(* CODESYS project tc2_bacnetrev12.library
   Company: Beckhoff Automation GmbH
   DefaultNamespace: Tc2_BACnetRev12
   Title: Tc2_BACnetRev12
   Description: The PLC library is a collection of function blocks for programming a BACnet controller. For each BACnet object function blocks are available that are read and written via the selected properties. In general a distinction is made between function blocks for server and client objects. Function blocks for client objects have the prefix "Remote", since they enable access to remote BACnet objects on other devices. The BACnet object function blocks ascertain whether process data are valid and the BACnet controller is ready for operation (bReady).
   Placeholder: Tc2_BACnetRev12
   Author: Beckhoff Automation
   Version: 2.4.3.0

Project tree, tasks and I/O mapping:
  libraries: Tc2_Standard, * (Beckhoff Automation GmbH); Tc2_System, * (Beckhoff Automation GmbH); Tc2_Utilities, * (Beckhoff Automation GmbH)
  Data types/
    BACnet Datatypes/
      [internal]/
        ADS/
          data type ST_BACnet_GlobalAdsBuffer
        CalendarEntry/
          data type E_BACnetCalendarEntryChoice
          data type E_BACnetCalendarEntryType
          data type ST_BACnet_CalendarEntryDate
          data type ST_BACnet_CalendarEntryDateRange
          data type ST_BACnet_CalendarEntryWeekNDay
        ExceptionSchedule/
          data type ST_BACnet_ExceptionScheduleCalDate
          data type ST_BACnet_ExceptionScheduleCalRef
          data type ST_BACnet_ExceptionScheduleCalWnD
        LogRecord/
          data type E_BACnetLogRecordChoice
          data type ST_BACnet_LogDatum
          data type ST_BACnet_LogDatumList
          data type ST_BACnet_LogRecord
          data type ST_BACnet_LogRecordList
        NotificationSink/
          data type ST_BACnet_NotificationSinkEventEntry
          data type ST_BACnet_NSinkEventValidFields
        Recipient/
          data type E_BACnetRecipientChoice
          data type ST_BACnet_DestinationDevice
          data type ST_BACnet_RecipientDevice
          data type T_BACnet_DestinationDeviceArray
        SpecialEvent/
          data type E_BACnetSpecialEventChoice
          data type ST_BACnet_SpecialEventCalendarEntryDate
          data type ST_BACnet_SpecialEventCalendarEntryRange
          data type ST_BACnet_SpecialEventCalendarEntryWnD
          data type ST_BACnet_SpecialEventCalendarReference
          data type ST_BACnet_SpecialEventListCalEntryDate
          data type ST_BACnet_SpecialEventListCalEntryRange
          data type ST_BACnet_SpecialEventListCalEntryWnD
          data type ST_BACnet_SpecialEventListCalReference
        WeeklySchedule/
          data type ST_BACnet_DailySchedule
        data type E_BACnetTimeStampChoice
        data type ST_BACnet_TimeStampDateTime
      [obsolete]/
        data type FB_BACnet_Accumulator_R9
        data type FB_BACnet_AnalogInput_R9
        data type FB_BACnet_AnalogOutput_R9
        data type FB_BACnet_AnalogValue_R9
        data type FB_BACnet_Averaging_R9
        data type FB_BACnet_BinaryInput_R9
        data type FB_BACnet_BinaryOutput_R9
        data type FB_BACnet_BinaryValue_R9
        data type FB_BACnet_Calendar_R9
        data type FB_BACnet_Command_R9
        data type FB_BACnet_Device_R9
        data type FB_BACnet_EventEnrollment_R9
        data type FB_BACnet_File_R9
        data type FB_BACnet_Group_R9
        data type FB_BACnet_Loop_R9
        data type FB_BACnet_MultiStateInput_R9
        data type FB_BACnet_MultiStateOutput_R9
        data type FB_BACnet_MultiStateValue_R9
        data type FB_BACnet_NotificationClass_R9
        data type FB_BACnet_Program_R9
        data type FB_BACnet_PulseConverter_R9
        data type FB_BACnet_Schedule_R9
        data type FB_BACnet_TrendLog_R9
      Diagnose/
        data type ST_BACnet_ConfirmedServiceDiag
        data type ST_BACnet_DiagEthStatistics
        data type ST_BACnet_DiagnosisTiming
        data type ST_BACnet_FrameStatistics
        data type ST_BACnet_Info
        data type ST_BACnet_ServerStatistics
        data type ST_BACnet_TcIoEthStatistic
        data type ST_BACnet_TcIoEthTxRxErrorCount
        data type ST_BACnet_UnConfirmedServiceDiag
      data type ST_BACnet_AdsConnection
      data type ST_BACnet_CharacterStringExt
      data type ST_BACnet_CharacterStringExtListEntry
      data type ST_BACnet_Date
      data type ST_BACnet_DateTime
      data type ST_BACnet_Diagnosis
      data type ST_BACnet_EventTransitionBits
      data type ST_BACnet_ExceptionScheduleBool
      data type ST_BACnet_ExceptionScheduleEntryBool
      data type ST_BACnet_ExceptionScheduleEntryReal
      data type ST_BACnet_ExceptionScheduleReal
      data type ST_BACnet_LimitEnable
      data type ST_BACnet_LogBufferEntryReal
      data type ST_BACnet_LogBufferReal
      data type ST_BACnet_NSinkEvent
      data type ST_BACnet_ObjectIdentifierList
      data type ST_BACnet_ObjectTypesSupported
      data type ST_BACnet_ProgramHandshakeRequests
      data type ST_BACnet_ProgramHandshakeStates
      data type ST_BACnet_RecipientListDevice
      data type ST_BACnet_RecipientListDeviceEntry
      data type ST_BACnet_ServicesSupported
      data type ST_BACnet_StatusFlags
      data type ST_BACnet_Time
      data type ST_BACnet_TimeValue
      data type ST_BACnet_TimeValueBool
      data type ST_BACnet_TimeValueList
      data type ST_BACnet_TimeValueReal
      data type ST_BACnet_Value
      data type ST_BACnet_WeeklyScheduleBool
      data type ST_BACnet_WeeklyScheduleReal
      data type T_BACnet_CalendarEntryTypeFilter
      data type T_BACnet_ObjectIdentifier
    BACnet Enumerations/
      data type E_BACNETACTION
      data type E_BACNETADAPTERSTATUS
      data type E_BACNETBINARYPV
      data type E_BACNETDATATYPES
      data type E_BACNETDAYSOFWEEKBITS
      data type E_BACNETDEVICESTATUS
      data type E_BACNETEVENTSTATE
      data type E_BACNETEVENTTRANSITIONBIT
      data type E_BACNETEVENTTYPE
      data type E_BACNETFILEACCESSMETHOD
      data type E_BACNETLIFESAFETYMODE
      data type E_BACNETLIFESAFETYOPERATION
      data type E_BACNETLIMITENABLEBITS
      data type E_BACNETLOGGINGTYPE
      data type E_BACNETLOOPMODE
      data type E_BACNETNOTIFYTYPE
      data type E_BACNETOBJECTSUPPORTEDBITS
      data type E_BACNETOBJECTTYPE
      data type E_BACNETPERSISTENTDATASTATE
      data type E_BACNETPIDTUNINGMODE
      data type E_BACNETPOLARITY
      data type E_BACNETPRIORITY
      data type E_BACNETPROGRAMERROR
      data type E_BACNETPROGRAMREQUEST
      data type E_BACNETPROGRAMSTATE
      data type E_BACNETPROPERTYIDENTIFIER
      data type E_BACNETRELIABILITY
      data type E_BACNETSEGMENTATION
      data type E_BACNETSERVICESSUPPORTEDBITS
      data type E_BACNETSILENCEDSTATE
      data type E_BACNETSTATUSFLAGS
      data type E_BACNETSTRINGENCODINGTYPES
      data type E_BACNETUNIT
  Global Variables/
    global variables BACnet_Globals
  POUs/
    [obsolete]/
      function F_GetVersionTcBACnet [ST]
    BACnet ADS/
      [obsolete]/
        function block FB_BACnet_NotificationSinkDelEntry [ST]
      Connection/
        function block _FB_BACnet_AdsConn [ST]
      Properties/
        Common/
          function block FB_BACnet_ReadProp [ST]
          function block FB_BACnet_WriteProp [ST]
        function block FB_BACnet_DescriptionProperty [ST]
        function block FB_BACnet_EventMessageTextsProperty [ST]: _NextEntry
        function block FB_BACnet_ExceptionScheduleProperty [ST]: _NextEvent, _NextTimeValue
        function block FB_BACnet_ExceptionSchedulePropertyReal [ST]: _NextEvent, _NextTimeValue
        function block FB_BACnet_LogBufferProperty [ST]: _NextLogDatum, _NextLogRecord
        function block FB_BACnet_ObjectListProperty [ST]
        function block FB_BACnet_ObjectNameProperty [ST]
        function block FB_BACnet_RecipientListProperty [ST]
        function block FB_BACnet_WeeklyScheduleProperty [ST]: _NextDay, _NextTimeValue
        function block FB_BACnet_WeeklySchedulePropertyReal [ST]: _NextDay, _NextTimeValue
      function block FB_BACnet_GetDiagInfo [ST]
      function block FB_BACnet_NSinkAcknEvent [ST]
      function block FB_BACnet_NSinkReadEvent [ST]
      function block FB_BACnet_NSinkRemoveEvent [ST]
      function block FB_BACnet_TimeSync [ST]
    BACnet Helper/
      [internal]/
        function _F_BACnet_AlignedSize [ST]
        function _F_BACnet_BitFieldBit [ST]
        function _F_BACnet_ChangeBitFieldBit [ST]
        function _F_BACnet_ChrStrExtLen [ST]
        function _F_BACnet_DecodeUCS2 [ST]
        function _F_BACnet_DecodeUCS4 [ST]
        function _F_BACnet_DecodeUTF8 [ST]
        function _F_BACnet_EncodeUTF8 [ST]
        function _F_BACnet_IsBitFieldBitSet [ST]
        function _F_BACnet_SetBitFieldBit [ST]
        function _F_BACnet_SysTimeDiff [ST]
        function _F_BACnet_UCS2ToWin1252 [ST]
        function _F_BACnet_UnSetBitFieldBit [ST]
        function _F_BACnet_Utf8ToWin1252 [ST]
        function _F_BACnet_Win1252ToUCS2 [ST]
        function _F_BACnet_Win1252ToUtf8 [ST]
        function block _FB_BACnet_PidTune [ST]
        function F_BACnet_AnalogPV [ST]
      DateTime/
        function F_BACnet_CheckDay [ST]
        function F_BACnet_CheckDayOfWeek [ST]
        function F_BACnet_CheckHour [ST]
        function F_BACnet_CheckHundredths [ST]
        function F_BACnet_CheckMinute [ST]
        function F_BACnet_CheckMonth [ST]
        function F_BACnet_CheckSecond [ST]
        function F_BACnet_CheckWeekOfMonth [ST]
        function F_BACnet_CheckYear [ST]
        function F_BACnet_DateHasPlaceholder [ST]
        function F_BACnet_DateMerge [ST]
        function F_BACnet_DateTime_TO_TimeStruct [ST]
        function F_BACnet_DateTimeString [ST]
        function F_BACnet_DateUnspecified [ST]
        function F_BACnet_DaysInMonth [ST]
        function F_BACnet_Get100msDate [ST]
        function F_BACnet_Get100msTime [ST]
        function F_BACnet_TimeHasPlaceholder [ST]
        function F_BACnet_TimeMerge [ST]
        function F_BACnet_TimeString [ST]
        function F_BACnet_TimeStruct_TO_DateTime [ST]
        function F_BACnet_TimeUnspecified [ST]
      Flags/
        function F_BACnet_EventTransitionFlags [ST]
        function F_BACnet_GetEventTransFlagsData [ST]
        function F_BACnet_GetLimitEnFlagsData [ST]
        function F_BACnet_GetStatusFlagsData [ST]
        function F_BACnet_LimitEnableFlags [ST]
        function F_BACnet_StatusFlags [ST]
      MultiState/
        function F_BACnet_MultiStatePV [ST]
      Real/
        function F_BACnet_IsFinite [ST]
        function F_BACnet_NAN [ST]
        function F_BACnet_RealEQ [ST]
        function F_BACnet_RealGE [ST]
        function F_BACnet_RealGT [ST]
        function F_BACnet_RealLE [ST]
        function F_BACnet_RealLT [ST]
        function F_BACnet_RealNothing [ST]
        function F_BACnet_RealNull [ST]
        function F_BACnet_RealPV [ST]
        function F_BACnet_RealToStr [ST]
      String/
        function F_BACnet_GetObjectIdString [ST]
        function block FB_BACnet_StringExtDecode [ST]
        function block FB_BACnet_StringExtEncode [ST]
      function F_BACnet_GetObjectListIndex [ST]
      function F_BACnet_GetObjId [ST]
      function F_BACnet_GetObjInstance [ST]
      function F_BACnet_GetObjType [ST]
      function block FB_BACnet_AccLimit [ST]
      function block FB_BACnet_AvgValue [ST]
      function block FB_BACnet_PidControl [ST]
      function block FB_BACnet_PT1 [ST]
    BACnet Logic/
      function F_BinPV_AND [ST]
      function F_BinPV_NOT [ST]
      function F_BinPV_OR [ST]
      function F_BinPV_To_Bool [ST]
      function F_BinPV_XOR [ST]
      function F_Bool_To_BinPV [ST]
    BACnet Objects/
      Local (Server)/
        [Internal]/
          function block _FB_BACnet_AnalogObject [ST]
          function block _FB_BACnet_BinaryObject [ST]
          function block _FB_BACnet_Object [ST]
        ADS/
          function block FB_BACnet_AnalogOutput_ADS [ST]
          function block FB_BACnet_AnalogValue_ADS [ST]
          function block FB_BACnet_BinaryOutput_ADS [ST]
          function block FB_BACnet_BinaryValue_ADS [ST]
          function block FB_BACnet_MultiStateOutput_ADS [ST]
          function block FB_BACnet_MultiStateValue_ADS [ST]
        DRV/
          function block FB_BACnet_Loop_DRV [ST]
          function block FB_BACnet_Loop_DRV_EX [ST]
        Extended Process Data/
          function block FB_BACnet_Accumulator_EX [ST]
          function block FB_BACnet_AnalogInput_EX [ST]
          function block FB_BACnet_AnalogOutput_EX [ST]
          function block FB_BACnet_AnalogValue_EX [ST]
          function block FB_BACnet_Averaging_EX [ST]
          function block FB_BACnet_BinaryInput_EX [ST]
          function block FB_BACnet_BinaryOutput_EX [ST]
          function block FB_BACnet_BinaryValue_EX [ST]
          function block FB_BACnet_Calendar_EX [ST]
          function block FB_BACnet_Command_EX [ST]
          function block FB_BACnet_EventEnrollment_EX [ST]
          function block FB_BACnet_File_EX [ST]
          function block FB_BACnet_Group_EX [ST]
          function block FB_BACnet_Loop_EX [ST]
          function block FB_BACnet_MultiStateInput_EX [ST]
          function block FB_BACnet_MultiStateOutput_EX [ST]
          function block FB_BACnet_MultiStateValue_EX [ST]
          function block FB_BACnet_NotificationClass_EX [ST]
          function block FB_BACnet_Program_EX [ST]
          function block FB_BACnet_PulseConverter_EX [ST]
          function block FB_BACnet_Schedule_EX [ST]
          function block FB_BACnet_TrendLog_EX [ST]
        R6/
          function block FB_BACnet_Accumulator_R6 [ST]
          function block FB_BACnet_Accumulator_RAW_R6 [ST]
        RAW/
          function block FB_BACnet_Accumulator_RAW [ST]
          function block FB_BACnet_AnalogInput_RAW [ST]
          function block FB_BACnet_AnalogOutput_RAW [ST]
          function block FB_BACnet_BinaryInput_RAW [ST]
          function block FB_BACnet_BinaryOutput_RAW [ST]
          function block FB_BACnet_MultiStateInput_RAW [ST]
          function block FB_BACnet_MultiStateOutput_RAW [ST]
          function block FB_BACnet_PulseConverter_RAW [ST]
        function block FB_BACnet_Accumulator [ST]
        function block FB_BACnet_AnalogInput [ST]
        function block FB_BACnet_AnalogOutput [ST]
        function block FB_BACnet_AnalogValue [ST]
        function block FB_BACnet_Averaging [ST]
        function block FB_BACnet_BinaryInput [ST]
        function block FB_BACnet_BinaryOutput [ST]
        function block FB_BACnet_BinaryValue [ST]
        function block FB_BACnet_Calendar [ST]
        function block FB_BACnet_Command [ST]
        function block FB_BACnet_Device [ST]
        function block FB_BACnet_EventEnrollment [ST]
        function block FB_BACnet_File [ST]
        function block FB_BACnet_Group [ST]
        function block FB_BACnet_Loop [ST]
        function block FB_BACnet_MultiStateInput [ST]
        function block FB_BACnet_MultiStateOutput [ST]
        function block FB_BACnet_MultiStateValue [ST]
        function block FB_BACnet_NotificationClass [ST]
        function block FB_BACnet_Program [ST]
        function block FB_BACnet_PulseConverter [ST]
        function block FB_BACnet_Schedule [ST]
        function block FB_BACnet_TrendLog [ST]
      Remote (Client)/
        Extended Process Data/
          function block FB_BACnet_RemoteAccumulator_EX [ST]
          function block FB_BACnet_RemoteAnalogInput_EX [ST]
          function block FB_BACnet_RemoteAnalogOutput_EX [ST]
          function block FB_BACnet_RemoteAnalogValue_EX [ST]
          function block FB_BACnet_RemoteAveraging_EX [ST]
          function block FB_BACnet_RemoteBinaryInput_EX [ST]
          function block FB_BACnet_RemoteBinaryOutput_EX [ST]
          function block FB_BACnet_RemoteBinaryValue_EX [ST]
          function block FB_BACnet_RemoteCalendar_EX [ST]
          function block FB_BACnet_RemoteCommand_EX [ST]
          function block FB_BACnet_RemoteEventEnrollment_EX [ST]
          function block FB_BACnet_RemoteFile_EX [ST]
          function block FB_BACnet_RemoteGroup_EX [ST]
          function block FB_BACnet_RemoteLoop_EX [ST]
          function block FB_BACnet_RemoteMultiStateInput_EX [ST]
          function block FB_BACnet_RemoteMultiStateOutput_EX [ST]
          function block FB_BACnet_RemoteMultiStateValue_EX [ST]
          function block FB_BACnet_RemoteNotificationClass_EX [ST]
          function block FB_BACnet_RemoteProgram_EX [ST]
          function block FB_BACnet_RemotePulseConverter_EX [ST]
          function block FB_BACnet_RemoteSchedule_EX [ST]
          function block FB_BACnet_RemoteTrendLog_EX [ST]
        WRITE/
          function block FB_BACnet_RemoteAnalogOutput_WR [ST]
          function block FB_BACnet_RemoteAnalogValue_WR [ST]
          function block FB_BACnet_RemoteBinaryOutput_WR [ST]
          function block FB_BACnet_RemoteBinaryValue_WR [ST]
          function block FB_BACnet_RemoteCommand_WR [ST]
          function block FB_BACnet_RemoteMultiStateOutput_WR [ST]
          function block FB_BACnet_RemoteMultiStateValue_WR [ST]
          function block FB_BACnet_RemoteProgram_WR [ST]
        function block FB_BACnet_RemoteAccumulator [ST]
        function block FB_BACnet_RemoteAnalogInput [ST]
        function block FB_BACnet_RemoteAnalogOutput [ST]
        function block FB_BACnet_RemoteAnalogValue [ST]
        function block FB_BACnet_RemoteAveraging [ST]
        function block FB_BACnet_RemoteBinaryInput [ST]
        function block FB_BACnet_RemoteBinaryOutput [ST]
        function block FB_BACnet_RemoteBinaryValue [ST]
        function block FB_BACnet_RemoteCalendar [ST]
        function block FB_BACnet_RemoteCommand [ST]
        function block FB_BACnet_RemoteDevice [ST]
        function block FB_BACnet_RemoteEventEnrollment [ST]
        function block FB_BACnet_RemoteFile [ST]
        function block FB_BACnet_RemoteGroup [ST]
        function block FB_BACnet_RemoteLoop [ST]
        function block FB_BACnet_RemoteMultiStateInput [ST]
        function block FB_BACnet_RemoteMultiStateOutput [ST]
        function block FB_BACnet_RemoteMultiStateValue [ST]
        function block FB_BACnet_RemoteNotificationClass [ST]
        function block FB_BACnet_RemoteProgram [ST]
        function block FB_BACnet_RemotePulseConverter [ST]
        function block FB_BACnet_RemoteSchedule [ST]
        function block FB_BACnet_RemoteTrendLog [ST]
    BACnet Signals/
      function block FB_BACnet_PWM [ST]
    function block FB_BACnet_Adapter [ST]: UpdateNetID
    function block FB_BACnet_NotificationSink [ST]
  Version/
    global variables Global_Version
*)

// Data types/BACnet Datatypes/[internal]/ADS/ST_BACnet_GlobalAdsBuffer
TYPE ST_BACnet_GlobalAdsBuffer :
STRUCT
	bTestSet	: BOOL;
	iLocked		: DINT; (* -1 Buffer not ready, 0 Buffer ready, 1..n Buffer used (locked) *)
	arrData		: ARRAY[0..BACnet_ADSBufferSize] OF BYTE;
END_STRUCT
END_TYPE

// Data types/BACnet Datatypes/[internal]/CalendarEntry/E_BACnetCalendarEntryChoice
TYPE E_BACnetCalendarEntryChoice :
(
(*
	BACnetDate              DATE;
	BACnetDateRange   		dateRange;
	BACnetWeekNDay          weekNDay;
*)
	BACnetCalendarEntryChoice_date,
	BACnetCalendarEntryChoice_dateRange,
	BACnetCalendarEntryChoice_weekNDay
);
END_TYPE

// Data types/BACnet Datatypes/[internal]/CalendarEntry/E_BACnetCalendarEntryType
TYPE E_BACnetCalendarEntryType : (* Not a BACnet-Stack type! *)
(
	BACnetCalendarEntryType_None,
	BACnetCalendarEntryType_Ref,
	BACnetCalendarEntryType_Date,
	BACnetCalendarEntryType_DateRange,
	BACnetCalendarEntryType_WeekNDay
);
END_TYPE

// Data types/BACnet Datatypes/[internal]/CalendarEntry/ST_BACnet_CalendarEntryDate
TYPE ST_BACnet_CalendarEntryDate :
STRUCT
(*
	typedef struct _BACnetCalendarEntry
	{
	      BACnetCalendarEntryChoice choice;
	      union
	      {
	            BACnetDate              date;
	            BACnetDateRange   dateRange;
	            BACnetWeekNDay          weekNDay;
	      };
	}BACnetCalendarEntry, *PBACnetCalendarEntry;
*)
	eEntryChoice		: E_BACnetCalendarEntryChoice;
	nRes				: WORD; (* ENUM alignment *)
	stDate				: ST_BACnet_Date;
END_STRUCT
END_TYPE

// Data types/BACnet Datatypes/[internal]/CalendarEntry/ST_BACnet_CalendarEntryDateRange
TYPE ST_BACnet_CalendarEntryDateRange :
STRUCT
(*
	typedef struct _BACnetCalendarEntry
	{
	      BACnetCalendarEntryChoice choice;
	      union
	      {
	            BACnetDate              date;
	            BACnetDateRange   dateRange;
	            BACnetWeekNDay          weekNDay;
	      };
	}BACnetCalendarEntry, *PBACnetCalendarEntry;
*)
	eEntryChoice		: E_BACnetCalendarEntryChoice;
	nRes				: WORD; (* ENUM alignment *)
	stStartDate			: ST_BACnet_Date;
	stEndDate			: ST_BACnet_Date;
END_STRUCT
END_TYPE

// Data types/BACnet Datatypes/[internal]/CalendarEntry/ST_BACnet_CalendarEntryWeekNDay
TYPE ST_BACnet_CalendarEntryWeekNDay :
STRUCT
(*
	typedef struct _BACnetCalendarEntry
	{
	      BACnetCalendarEntryChoice choice;
	      union
	      {
	            BACnetDate              date;
	            BACnetDateRange   dateRange;
	            BACnetWeekNDay          weekNDay;
	      };
	}BACnetCalendarEntry, *PBACnetCalendarEntry;
*)
	eEntryChoice	: E_BACnetCalendarEntryChoice;
	nRes1			: WORD; (* ENUM alignment *)
	iMonth			: USINT;
	iWeekOfMonth	: USINT;
	iDay			: USINT;
	nRes2			: USINT; (* weekNDay alignment *)
END_STRUCT
END_TYPE

// Data types/BACnet Datatypes/[internal]/ExceptionSchedule/ST_BACnet_ExceptionScheduleCalDate
TYPE ST_BACnet_ExceptionScheduleCalDate :
STRUCT
	stStart			: ST_BACnet_Date;
	stEnd			: ST_BACnet_Date;
END_STRUCT
END_TYPE

// Data types/BACnet Datatypes/[internal]/ExceptionSchedule/ST_BACnet_ExceptionScheduleCalRef
TYPE ST_BACnet_ExceptionScheduleCalRef :
STRUCT
	tCalObjectId	: T_BACnet_ObjectIdentifier := 16#FFFFFFFF;
END_STRUCT
END_TYPE

// Data types/BACnet Datatypes/[internal]/ExceptionSchedule/ST_BACnet_ExceptionScheduleCalWnD
TYPE ST_BACnet_ExceptionScheduleCalWnD :
STRUCT
	iMonth			: USINT; (* 255 = all months of year *)
	iWeekOfMonth	: USINT; (* 255 = all weeks of month *)
	iDay			: USINT; (* 255 = all days of month *)
END_STRUCT
END_TYPE

// Data types/BACnet Datatypes/[internal]/LogRecord/E_BACnetLogRecordChoice
TYPE E_BACnetLogRecordChoice :
(
(*
enum BACnetLogRecordChoice
{
      logStatus,              // [0] BACnetLogStatus,
      booleanValue,           // [1] BOOL,
      realValue,              // [2] REAL,
      enumValue,              // [3] ENUMERATED, __ Optionally limited to 32 bits
      unsignedValue,          // [4] Unsigned, __ Optionally limited to 32 bits
      signedValue,            // [5] INTEGER, __ Optionally limited to 32 bits
      bitstringValue,         // [6] BIT STRING, __ Optionally limited to 32 bits
      nullValue,              // [7] NULL,
      failure,                // [8] Error,
      timeChange,             // [9] REAL,
      anyValue,               // [10] ABSTRACT_SYNTAX.&Type __ Optional
};
*)
	BACnetLogRecordChoice_logStatus 	:= 0, (* BACnetLogStatus *)
	BACnetLogRecordChoice_booleanValue := 1, (*  BOOL, *)
	BACnetLogRecordChoice_realValue	:= 2, (*  REAL, *)
	BACnetLogRecordChoice_enumValue	:= 3, (*  ENUMERATED, __ Optionally limited TO 32 bits *)
	BACnetLogRecordChoice_unsignedValue:= 4, (*  Unsigned, __ Optionally limited TO 32 bits *)
	BACnetLogRecordChoice_signedValue	:= 5, (*  INTEGER, __ Optionally limited TO 32 bits *)
	BACnetLogRecordChoice_bitstringValue:= 6, (*  BIT STRING, __ Optionally limited TO 32 bits *)
	BACnetLogRecordChoice_nullValue	:= 7, (*  NULL, *)
	BACnetLogRecordChoice_failure		:= 8, (*  Error, *)
	BACnetLogRecordChoice_timeChange	:= 9, (*  REAL, *)
	BACnetLogRecordChoice_anyValue		:= 10 (*  ABSTRACT_SYNTAX.&TYPE __ Optional *)
);
END_TYPE

// Data types/BACnet Datatypes/[internal]/LogRecord/ST_BACnet_LogDatum
TYPE ST_BACnet_LogDatum :
STRUCT
(*

typedef struct _BACnetLogDatum
{
      BACnetLogRecordChoice choice;
      union
      {
            DWORD logStatus; // BitString ... of type BACnetLogStatus
            BOOL booleanValue;
            FLOAT realValue;
            EnumerationValueType enumerationValue;
            ULONG unsignedValue;
            DWORD signedValue;
            DWORD bitstringValue;
            DWORD nullValue;
            BACnetError failure; 
            FLOAT timeChange;
            AnyType anyValue; // ABSTRACT-SYNTAX.&Type
      };
}BACnetLogDatum, *PBACnetLogDatum;

*)
	choice	: E_BACnetLogRecordChoice;
	nRes	: WORD; (* ENUM alignment to 4 byte *)
	nData	: ARRAY[0..4] OF DWORD; (* 20 byte min. size - data type depending on choice selection *)
END_STRUCT
END_TYPE

// Data types/BACnet Datatypes/[internal]/LogRecord/ST_BACnet_LogDatumList
TYPE ST_BACnet_LogDatumList :
STRUCT
(*

typedef struct _BACnetLogDatumList
{
      DWORD nEntrySize; // 0x80000000 -> next entry
      DWORD reserved;
      BACnetLogDatum listEntry;
}BACnetLogDatumList, *PBACnetLogDatumList;

*)
	nEntrySize	: DWORD; (* 0x80000000 -> next entry *)
	reserved	: DWORD;
	listEntry	: ST_BACnet_LogDatum; (* first entry of log datum list *)
END_STRUCT
END_TYPE

// Data types/BACnet Datatypes/[internal]/LogRecord/ST_BACnet_LogRecord
TYPE ST_BACnet_LogRecord :
STRUCT
(*

typedef STRUCT _BACnetLogRecord
{
      ULONG validFields;
      BACnetDateTime timestamp;          // [0]
      DWORD statusFlags;                       // [2] optional
      BACnetLogDatumList logDatum;  // [1]
}BACnetLogRecord, *PBACnetLogRecord;

*)
	validFields	: UDINT;
	timestamp	: ST_BACnet_DateTime;
	statusFlags	: DWORD;
	logDatum	: ST_BACnet_LogDatumList;
END_STRUCT
END_TYPE

// Data types/BACnet Datatypes/[internal]/LogRecord/ST_BACnet_LogRecordList
TYPE ST_BACnet_LogRecordList :
STRUCT
(*

typedef struct _BACnetLogRecordList
{
      DWORD nEntrySize; // 0x80000000 -> next entry
      DWORD nSequence;  // "reserved"     -> Number of Sequence begins with 1
      BACnetLogRecord listEntry;
}BACnetLogRecordList, *PBACnetLogRecordList;

*)
	nEntrySize	: DWORD; (* 16#80000000 -> next entry *)
	nSequence	: DWORD; (* "reserved"  -> Number OF Sequence begins with 1 *)
	listEntry	: ST_BACnet_LogRecord; (* first entry of record list *)
END_STRUCT
END_TYPE

// Data types/BACnet Datatypes/[internal]/NotificationSink/ST_BACnet_NotificationSinkEventEntry
TYPE ST_BACnet_NotificationSinkEventEntry :
STRUCT
	_fillBytes00				: ARRAY[0..7] OF BYTE; (* list header *)
	validFields					: UDINT;	(*	ULONG validFields; *)
	processIdentifier			: UDINT; (*     ULONG processIdentifier; *)
	initiatingDeviceIdentifier	: T_BACnet_ObjectIdentifier; (*  BACnetObjectIdentifier initiatingDeviceIdentifier; *)
	eventObjectIdentifier		: T_BACnet_ObjectIdentifier; (*  BACnetObjectIdentifier eventObjectIdentifier; *)
	timeStamp					: ST_BACnet_TimeStampDateTime;   (* BACnetTimeStamp timeStamp; *)
	notificationClass			: UDINT;  (* ULONG notificationClass;*)
	priority					: UDINT;  (* ULONG priority; *)
	eventType					: E_BACNETEVENTTYPE; (*  BACnetEventType eventType; *)
	_fillBytes01				: WORD; (* fill bytes *)
	messageText					: ARRAY[1..BACnet_STRING_MAXLENGTH] OF BYTE;
	notifyType					: E_BACNETNOTIFYTYPE;  (* BACnetNotifyType notifyType; *)
	_fillBytes02				: WORD; (* fill bytes *)
	ackRequired					: BOOL; (*  BOOL ackRequired; *)
	_fillBytes03				: ARRAY[0..2] OF BYTE; (* fill bytes *)
	fromState					: E_BACNETEVENTSTATE; (*   BACnetEventState fromState; *)
	_fillBytes04				: WORD; (* fill bytes *)
	toState						: E_BACNETEVENTSTATE; (*  BACnetEventState toState; *)
	_fillBytes05				: WORD; (* fill bytes *)
	eventParameterRaw			: ARRAY[0..127] OF BYTE; (* PBACnetNotificationParameters pEventValues; *)
END_STRUCT
END_TYPE

// Data types/BACnet Datatypes/[internal]/NotificationSink/ST_BACnet_NSinkEventValidFields
TYPE ST_BACnet_NSinkEventValidFields :
STRUCT
      bProcessIdentifier:BOOL; (* Bit0 *)
      bInitiatingDeviceIdentifier:BOOL; (* Bit1 *)
      bEventObjectIdentifier:BOOL; (* Bit2 *)
      bTimeStamp:BOOL; (* Bit3 *)
      bNotificationClass:BOOL; (* Bit4 *)
      bPriority:BOOL; (* Bit5 *)
      bEventType:BOOL; (* Bit6 *)
      bMessageText:BOOL; (* Bit7 *)
      bNotifyType:BOOL; (* Bit8 *)
      bAckRequired:BOOL; (* Bit9 *)
      bFromState:BOOL; (* Bit10 *)
      bToState:BOOL; (* Bit11 *)
      bEventValues:BOOL; (* Bit12 *)
END_STRUCT
END_TYPE

// Data types/BACnet Datatypes/[internal]/Recipient/E_BACnetRecipientChoice
TYPE E_BACnetRecipientChoice :
(
	BACnetRecipientChoice_device,
	BACnetRecipientChoice_address
);
END_TYPE

// Data types/BACnet Datatypes/[internal]/Recipient/ST_BACnet_DestinationDevice
TYPE ST_BACnet_DestinationDevice :
STRUCT
	nValidDaysFlags	: DWORD; (* Bit: 9 = Sunday, 10 = Saturday, 11 = Friday, 12 = Thursday, 13 = Wednesday, 14 = Tuesday, 15 = Monday *)
	stFromTime		: ST_BACnet_Time;
	stToTime		: ST_BACnet_Time;
	stRecipient		: ST_BACnet_RecipientDevice;
	res1			: ARRAY[0..11] OF BYTE; (* allignment *)
	nProcessId		: UDINT;
	nEventTransBits	: DWORD; (* Bit: 12 = to_offnormal, 13 = to_fault, 14 = to_normal *)
	bIssueConfNot	: BOOL;
	res2			: ARRAY[0..2] OF BYTE; (* allignment *)
END_STRUCT
END_TYPE

// Data types/BACnet Datatypes/[internal]/Recipient/ST_BACnet_RecipientDevice
TYPE ST_BACnet_RecipientDevice :
STRUCT
	eRecipientChoice: E_BACnetRecipientChoice;
	res				: WORD; (* allignment *)
	tDeviceId		: T_BACnet_ObjectIdentifier := 16#FFFFFFFF;
END_STRUCT
END_TYPE

// Data types/BACnet Datatypes/[internal]/Recipient/T_BACnet_DestinationDeviceArray
TYPE T_BACnet_DestinationDeviceArray : ARRAY[0..BACnet_MaxDestinationArray] OF ST_BACnet_DestinationDevice; END_TYPE

// Data types/BACnet Datatypes/[internal]/SpecialEvent/E_BACnetSpecialEventChoice
TYPE E_BACnetSpecialEventChoice :
(
(*
	enum BACnetSpecialEventChoice
	{
	      calendarEntry,
	      calendarReference,
	      MaxBACnetSpecialEventChoice
	};
*)
	BACnetSpecialEventChoice_calendarEntry,
	BACnetSpecialEventChoice_calendarReference
);
END_TYPE

// Data types/BACnet Datatypes/[internal]/SpecialEvent/ST_BACnet_SpecialEventCalendarEntryDate
TYPE ST_BACnet_SpecialEventCalendarEntryDate :
STRUCT
(*
	typedef struct _BACnetSpecialEvent
	{
	      BACnetSpecialEventChoice choice;
	      union
	      {
	            BACnetCalendarEntry calendarEntry;
	            BACnetObjectIdentifier calendarReference;
	      };
	      DWORD eventPriority; // DWORD due to alignment
	      DWORD reserved;
	      BACnetTimeValueList listOfTimeValues;
	}BACnetSpecialEvent, *PBACnetSpecialEvent;
*)

	eEventChoice		: E_BACnetSpecialEventChoice;
	nRes1				: WORD; (* ENUM alignment *)
	stCalEntry			: ST_BACnet_CalendarEntryDate;
	nRes2				: DWORD;
	iEventPriority		: DWORD;
	nRes3				: DWORD;
	stListOfTimeValues	: ST_BACnet_TimeValueList;

END_STRUCT
END_TYPE

// Data types/BACnet Datatypes/[internal]/SpecialEvent/ST_BACnet_SpecialEventCalendarEntryRange
TYPE ST_BACnet_SpecialEventCalendarEntryRange :
STRUCT
(*
	typedef struct _BACnetSpecialEvent
	{
	      BACnetSpecialEventChoice choice;
	      union
	      {
	            BACnetCalendarEntry calendarEntry;
	            BACnetObjectIdentifier calendarReference;
	      };
	      DWORD eventPriority; // DWORD due to alignment
	      DWORD reserved;
	      BACnetTimeValueList listOfTimeValues;
	}BACnetSpecialEvent, *PBACnetSpecialEvent;
*)

	eEventChoice		: E_BACnetSpecialEventChoice;
	nRes1				: WORD; (* ENUM alignment *)
	stCalEntry			: ST_BACnet_CalendarEntryDateRange;
	iEventPriority		: DWORD;
	nRes2				: DWORD;
	stListOfTimeValues	: ST_BACnet_TimeValueList;

END_STRUCT
END_TYPE

// Data types/BACnet Datatypes/[internal]/SpecialEvent/ST_BACnet_SpecialEventCalendarEntryWnD
TYPE ST_BACnet_SpecialEventCalendarEntryWnD :
STRUCT
(*
	typedef struct _BACnetSpecialEvent
	{
	      BACnetSpecialEventChoice choice;
	      union
	      {
	            BACnetCalendarEntry calendarEntry;
	            BACnetObjectIdentifier calendarReference;
	      };
	      DWORD eventPriority; // DWORD due to alignment
	      DWORD reserved;
	      BACnetTimeValueList listOfTimeValues;
	}BACnetSpecialEvent, *PBACnetSpecialEvent;
*)

	eEventChoice		: E_BACnetSpecialEventChoice;
	nRes1				: WORD; (* ENUM alignment *)
	stCalEntry			: ST_BACnet_CalendarEntryWeekNDay;
	nRes2				: DWORD;
	iEventPriority		: DWORD;
	nRes3				: DWORD;
	stListOfTimeValues	: ST_BACnet_TimeValueList;

END_STRUCT
END_TYPE

// Data types/BACnet Datatypes/[internal]/SpecialEvent/ST_BACnet_SpecialEventCalendarReference
TYPE ST_BACnet_SpecialEventCalendarReference :
STRUCT
(*
	typedef struct _BACnetSpecialEvent
	{
	      BACnetSpecialEventChoice choice;
	      union
	      {
	            BACnetCalendarEntry calendarEntry;
	            BACnetObjectIdentifier calendarReference;
	      };
	      DWORD eventPriority; // DWORD due to alignment
	      DWORD reserved;
	      BACnetTimeValueList listOfTimeValues;
	}BACnetSpecialEvent, *PBACnetSpecialEvent;
*)

	eEventChoice		: E_BACnetSpecialEventChoice;
	nRes1				: WORD; (* ENUM alignment *)
	tCalRef				: T_BACnet_ObjectIdentifier := 16#FFFFFFFF;
	nRes2				: DWORD;
	nRes3				: DWORD;
	iEventPriority		: DWORD;
	nRes4				: DWORD;
	stListOfTimeValues	: ST_BACnet_TimeValueList;

END_STRUCT
END_TYPE

// Data types/BACnet Datatypes/[internal]/SpecialEvent/ST_BACnet_SpecialEventListCalEntryDate
TYPE ST_BACnet_SpecialEventListCalEntryDate :
STRUCT
(*
	typedef struct _BACnetSpecialEventList
	{
	      DWORD nEntrySize; // 0x80000000 -> next entry
	      DWORD reserved;
	      BACnetSpecialEvent listEntry;
	}BACnetSpecialEventList, *PBACnetSpecialEventList;
*)
	nEntrySize		: DWORD;
	nRes			: DWORD;
	stListEntry		: ST_BACnet_SpecialEventCalendarEntryDate;
END_STRUCT
END_TYPE

// Data types/BACnet Datatypes/[internal]/SpecialEvent/ST_BACnet_SpecialEventListCalEntryRange
TYPE ST_BACnet_SpecialEventListCalEntryRange :
STRUCT
(*
	typedef struct _BACnetSpecialEventList
	{
	      DWORD nEntrySize; // 0x80000000 -> next entry
	      DWORD reserved;
	      BACnetSpecialEvent listEntry;
	}BACnetSpecialEventList, *PBACnetSpecialEventList;
*)
	nEntrySize		: DWORD;
	nRes			: DWORD;
	stListEntry		: ST_BACnet_SpecialEventCalendarEntryRange;
END_STRUCT
END_TYPE

// Data types/BACnet Datatypes/[internal]/SpecialEvent/ST_BACnet_SpecialEventListCalEntryWnD
TYPE ST_BACnet_SpecialEventListCalEntryWnD :
STRUCT
(*
	typedef struct _BACnetSpecialEventList
	{
	      DWORD nEntrySize; // 0x80000000 -> next entry
	      DWORD reserved;
	      BACnetSpecialEvent listEntry;
	}BACnetSpecialEventList, *PBACnetSpecialEventList;
*)
	nEntrySize		: DWORD;
	nRes			: DWORD;
	stListEntry		: ST_BACnet_SpecialEventCalendarEntryWnD;
END_STRUCT
END_TYPE

// Data types/BACnet Datatypes/[internal]/SpecialEvent/ST_BACnet_SpecialEventListCalReference
TYPE ST_BACnet_SpecialEventListCalReference :
STRUCT
(*
	typedef struct _BACnetSpecialEventList
	{
	      DWORD nEntrySize; // 0x80000000 -> next entry
	      DWORD reserved;
	      BACnetSpecialEvent listEntry;
	}BACnetSpecialEventList, *PBACnetSpecialEventList;
*)
	nEntrySize		: DWORD;
	nRes			: DWORD;
	stListEntry		: ST_BACnet_SpecialEventCalendarReference;
END_STRUCT
END_TYPE

// Data types/BACnet Datatypes/[internal]/WeeklySchedule/ST_BACnet_DailySchedule
TYPE ST_BACnet_DailySchedule :
STRUCT
(*
	PropWeeklySchedule:
	
	typedef struct _BACnetDailySchedule
	{
	      DWORD nEntrySize; // 0x80000000 -> next entry
	      DWORD reserved;
	      BACnetTimeValueList listEntry;
	} BACnetDailySchedule, *PBACnetDailySchedule;
*)
	nEntrySize	: DWORD;
	nRes		: DWORD;
	stListEntry	: ST_BACnet_TimeValueList;
END_STRUCT
END_TYPE

// Data types/BACnet Datatypes/[internal]/E_BACnetTimeStampChoice
TYPE E_BACnetTimeStampChoice :
(
	BACnetTimeStampChoice_ts_time,
    BACnetTimeStampChoice_sequenceNumber,
    BACnetTimeStampChoice_dateTime
);
END_TYPE

// Data types/BACnet Datatypes/[internal]/ST_BACnet_TimeStampDateTime
TYPE ST_BACnet_TimeStampDateTime :
STRUCT
	eType		: E_BACnetTimeStampChoice;
	_fillBytes	: WORD;
	stDateTime	: ST_BACnet_DateTime;
END_STRUCT
END_TYPE

// Data types/BACnet Datatypes/[obsolete]/FB_BACnet_Accumulator_R9
TYPE FB_BACnet_Accumulator_R9 : FB_BACnet_Accumulator;
END_TYPE

// Data types/BACnet Datatypes/[obsolete]/FB_BACnet_AnalogInput_R9
TYPE FB_BACnet_AnalogInput_R9 : FB_BACnet_AnalogInput;
END_TYPE

// Data types/BACnet Datatypes/[obsolete]/FB_BACnet_AnalogOutput_R9
TYPE FB_BACnet_AnalogOutput_R9 : FB_BACnet_AnalogOutput;
END_TYPE

// Data types/BACnet Datatypes/[obsolete]/FB_BACnet_AnalogValue_R9
TYPE FB_BACnet_AnalogValue_R9 : FB_BACnet_AnalogValue;
END_TYPE

// Data types/BACnet Datatypes/[obsolete]/FB_BACnet_Averaging_R9
TYPE FB_BACnet_Averaging_R9 : FB_BACnet_Averaging;
END_TYPE

// Data types/BACnet Datatypes/[obsolete]/FB_BACnet_BinaryInput_R9
TYPE FB_BACnet_BinaryInput_R9 : FB_BACnet_BinaryInput;
END_TYPE

// Data types/BACnet Datatypes/[obsolete]/FB_BACnet_BinaryOutput_R9
TYPE FB_BACnet_BinaryOutput_R9 : FB_BACnet_BinaryOutput;
END_TYPE

// Data types/BACnet Datatypes/[obsolete]/FB_BACnet_BinaryValue_R9
TYPE FB_BACnet_BinaryValue_R9 : FB_BACnet_BinaryValue;
END_TYPE

// Data types/BACnet Datatypes/[obsolete]/FB_BACnet_Calendar_R9
TYPE FB_BACnet_Calendar_R9 : FB_BACnet_Calendar;
END_TYPE

// Data types/BACnet Datatypes/[obsolete]/FB_BACnet_Command_R9
TYPE FB_BACnet_Command_R9 : FB_BACnet_Command;
END_TYPE

// Data types/BACnet Datatypes/[obsolete]/FB_BACnet_Device_R9
TYPE FB_BACnet_Device_R9 : FB_BACnet_Device;
END_TYPE

// Data types/BACnet Datatypes/[obsolete]/FB_BACnet_EventEnrollment_R9
TYPE FB_BACnet_EventEnrollment_R9 : FB_BACnet_EventEnrollment;
END_TYPE

// Data types/BACnet Datatypes/[obsolete]/FB_BACnet_File_R9
TYPE FB_BACnet_File_R9 : FB_BACnet_File;
END_TYPE

// Data types/BACnet Datatypes/[obsolete]/FB_BACnet_Group_R9
TYPE FB_BACnet_Group_R9 : FB_BACnet_Group;
END_TYPE

// Data types/BACnet Datatypes/[obsolete]/FB_BACnet_Loop_R9
TYPE FB_BACnet_Loop_R9 : FB_BACnet_Loop;
END_TYPE

// Data types/BACnet Datatypes/[obsolete]/FB_BACnet_MultiStateInput_R9
TYPE FB_BACnet_MultiStateInput_R9 : FB_BACnet_MultiStateInput;
END_TYPE

// Data types/BACnet Datatypes/[obsolete]/FB_BACnet_MultiStateOutput_R9
TYPE FB_BACnet_MultiStateOutput_R9 : FB_BACnet_MultiStateOutput;
END_TYPE

// Data types/BACnet Datatypes/[obsolete]/FB_BACnet_MultiStateValue_R9
TYPE FB_BACnet_MultiStateValue_R9 : FB_BACnet_MultiStateValue;
END_TYPE

// Data types/BACnet Datatypes/[obsolete]/FB_BACnet_NotificationClass_R9
TYPE FB_BACnet_NotificationClass_R9 : FB_BACnet_NotificationClass;
END_TYPE

// Data types/BACnet Datatypes/[obsolete]/FB_BACnet_Program_R9
TYPE FB_BACnet_Program_R9 : FB_BACnet_Program;
END_TYPE

// Data types/BACnet Datatypes/[obsolete]/FB_BACnet_PulseConverter_R9
TYPE FB_BACnet_PulseConverter_R9 : FB_BACnet_PulseConverter;
END_TYPE

// Data types/BACnet Datatypes/[obsolete]/FB_BACnet_Schedule_R9
TYPE FB_BACnet_Schedule_R9 : FB_BACnet_Schedule;
END_TYPE

// Data types/BACnet Datatypes/[obsolete]/FB_BACnet_TrendLog_R9
TYPE FB_BACnet_TrendLog_R9 : FB_BACnet_TrendLog;
END_TYPE

// Data types/BACnet Datatypes/Diagnose/ST_BACnet_ConfirmedServiceDiag
TYPE ST_BACnet_ConfirmedServiceDiag :
STRUCT
	nReqSend: DWORD; (* ULONG *)
	nReqSendFail: DWORD; (* ULONG *)
	nReqRecv: DWORD; (* ULONG *)
	nReqRecvFail: DWORD; (* ULONG *)
	nAckSend: DWORD; (* ULONG *)
	nAckSendFail: DWORD; (* ULONG *)
	nAckRecv: DWORD; (* ULONG *)
	nAckRecvFail: DWORD; (* ULONG *)
END_STRUCT
END_TYPE

// Data types/BACnet Datatypes/Diagnose/ST_BACnet_DiagEthStatistics
TYPE ST_BACnet_DiagEthStatistics :
STRUCT
	ethStat: ST_BACnet_TcIoEthStatistic;
	txRxErrCnt: ST_BACnet_TcIoEthTxRxErrorCount;
END_STRUCT
END_TYPE

// Data types/BACnet Datatypes/Diagnose/ST_BACnet_DiagnosisTiming
TYPE ST_BACnet_DiagnosisTiming :
STRUCT
	msIoInCurExecutionTime: DWORD; (* ULONG *)
	msIoInMinExecutionTime: DWORD; (* ULONG *)
	msIoInMaxExecutionTime: DWORD; (* ULONG *)
	msIoOutCurExecutionTime: DWORD; (* ULONG *)
	msIoOutMinExecutionTime: DWORD; (* ULONG *)
	msIoOutMaxExecutionTime: DWORD; (* ULONG *)
	msCycleCurExecutionTime: DWORD; (* ULONG *)
	msCycleMinExecutionTime: DWORD; (* ULONG *)
	msCycleMaxExecutionTime: DWORD; (* ULONG *)
	msInputCurDistanceTime: DWORD; (* ULONG *)
	msInputMinDistanceTime: DWORD; (* ULONG *)
	msInputMaxDistanceTime: DWORD; (* ULONG *)
END_STRUCT
END_TYPE

// Data types/BACnet Datatypes/Diagnose/ST_BACnet_FrameStatistics
TYPE ST_BACnet_FrameStatistics :
STRUCT
	confirmed: ARRAY[0..29] OF ST_BACnet_ConfirmedServiceDiag; (* [SERVICE_CONFIRMED_MAX + 1]; 29 + 1 *)
	unConfirmed: ARRAY[0..9] OF ST_BACnet_UnConfirmedServiceDiag; (* [SERVICE_UNCONFIRMED_MAX + 1]; 9 *)
	nSegmSendTimeouts: DWORD; (* ULONG *)
	nFrameAllocFailCnt: DWORD; (* ULONG *)
	nFrameSendCnt: DWORD; (* ULONG *)
	nFrameSendFailCnt: DWORD; (* ULONG *)
	nFrameRecvCnt: DWORD; (* ULONG *)
	nFrameRecvFailCnt: DWORD; (* ULONG *)
	nLinkStatusChangedCnt: DWORD; (* ULONG *)
END_STRUCT
END_TYPE

// Data types/BACnet Datatypes/Diagnose/ST_BACnet_Info
TYPE ST_BACnet_Info :
STRUCT
	nAmsAllocCnt: DINT; (* LONG *)
	nAmsAllocCntMax: DWORD; (* ULONG *)
	nAmsAllocFailCnt: DWORD; (* ULONG *)
	nAvailPhysMemBytes: DWORD; (* ULONG *)
	nAvailFlashMemBytes: ARRAY[0..1] OF DWORD; (* ULONGLONG *)
	nRecvFrameFifoSize: DWORD; (* ULONG *)
	nEmptyFrameFifoSize: DWORD; (* ULONG *)
	nRecvSegmUDPFramesListSize: DWORD; (* ULONG *)
	nRecvSegmFramesListSize: DWORD; (* ULONG *)
	nSendSegmFramesListSize: DWORD; (* ULONG *)
	nClientScanListSize: DWORD; (* ULONG *)
	nAmsRecvMissCount: DWORD; (* ULONG *)
END_STRUCT
END_TYPE

// Data types/BACnet Datatypes/Diagnose/ST_BACnet_ServerStatistics
TYPE ST_BACnet_ServerStatistics :
STRUCT
	nOpenRequests: DWORD; (* ULONG *)
	nRequestRetries: DWORD; (* ULONG *)
	nRequestTimeOuts: DWORD; (* ULONG *)
	nPropChanges: DWORD; (* ULONG *)
	nPersistWrites: DWORD; (* ULONG *)
	persistChangeSetId: DWORD; (* ULONG *)
	secpersistNextWrite: DWORD; (* ULONG *)
	persistLastWrite: ST_BACnet_DateTime;
END_STRUCT
END_TYPE

// Data types/BACnet Datatypes/Diagnose/ST_BACnet_TcIoEthStatistic
TYPE ST_BACnet_TcIoEthStatistic :
STRUCT
	dcTimeStamp: ARRAY[0..1] OF DWORD; (* ULONGLONG *)
	sendFrames: DWORD; (* ULONG *)
	recvFrames: DWORD; (* ULONG *)
	sendTimeRTime: DWORD; (* ULONG *)
	recvTimeRTime: DWORD; (* ULONG *)
	sendTimeNdis: DWORD; (* ULONG *)
	recvTimeNdis: DWORD; (* ULONG *)
END_STRUCT
END_TYPE

// Data types/BACnet Datatypes/Diagnose/ST_BACnet_TcIoEthTxRxErrorCount
TYPE ST_BACnet_TcIoEthTxRxErrorCount :
STRUCT
	txCnt: DWORD; (* ULONG *)
	rxCnt: DWORD; (* ULONG *)
END_STRUCT
END_TYPE

// Data types/BACnet Datatypes/Diagnose/ST_BACnet_UnConfirmedServiceDiag
TYPE ST_BACnet_UnConfirmedServiceDiag :
STRUCT
	nReqSend: DWORD; (* ULONG *)
	nReqSendFail: DWORD; (* ULONG *)
	nReqRecv: DWORD; (* ULONG *)
	nReqRecvFail: DWORD; (* ULONG *)
END_STRUCT
END_TYPE

// Data types/BACnet Datatypes/ST_BACnet_AdsConnection
TYPE ST_BACnet_AdsConnection :
STRUCT
	bValid		: BOOL; (* information are valid *)
	nReload		: USINT; (* reload counter *)
	sAmsNetId	: T_AmsNetId;
	nAmsPort	: T_AmsPort := 1000;
	bServer		: BOOL;
	bClient		: BOOL;
	bNSink		: BOOL;
	nDeviceId	: UDINT; (* Device object instance resp. BACnet ID *)
END_STRUCT
END_TYPE

// Data types/BACnet Datatypes/ST_BACnet_CharacterStringExt
TYPE ST_BACnet_CharacterStringExt :
STRUCT
	cookie		: BYTE; (* 0 -> DO differentiate normal strings *)
	encoding	: BYTE;
	strLen		: UINT;
	stringData	: ARRAY[1..BACnet_STRING_MAXLENGTH] OF BYTE;
END_STRUCT
END_TYPE

// Data types/BACnet Datatypes/ST_BACnet_CharacterStringExtListEntry
TYPE ST_BACnet_CharacterStringExtListEntry :
STRUCT
(* list header *)
	nEntrySize	: DWORD; (* byte size of data *)
	hdrInfo		: DWORD;
(* data *)
	extString	: ST_BACnet_CharacterStringExt;
END_STRUCT
END_TYPE

// Data types/BACnet Datatypes/ST_BACnet_Date
TYPE ST_BACnet_Date :
STRUCT
	nYear		: BYTE := 16#FF; (* year minus 1900 X'FF' = unspecified *)
	nMonth		: BYTE := 16#FF; (* (1.. 12) 1 = January X'FF' = unspecified *)
	nDay		: BYTE := 16#FF;	(* day OF month (1..31), X'FF' = unspecified *)
	nDayOfWeek	: BYTE := 16#FF;	(* day OF week (1..7) 1 = Monday -- 7 = Sunday -- X'FF' = unspecified *)
END_STRUCT
END_TYPE

// Data types/BACnet Datatypes/ST_BACnet_DateTime
TYPE ST_BACnet_DateTime :
STRUCT
	stDate		: ST_BACnet_Date;
	stTime		: ST_BACnet_Time;
END_STRUCT
END_TYPE

// Data types/BACnet Datatypes/ST_BACnet_Diagnosis
TYPE ST_BACnet_Diagnosis :
STRUCT
	ethDevice: ST_BACnet_DiagEthStatistics;
	execTiming: ST_BACnet_DiagnosisTiming;
	frameStatistics: ST_BACnet_FrameStatistics;
	nRes1 : DWORD;
	info: ST_BACnet_Info;
	nRes2 : DWORD;
	serverInfo: ST_BACnet_ServerStatistics;
	lastUpdate: ST_BACnet_DateTime;
	nRes3 : DWORD;
END_STRUCT
END_TYPE

// Data types/BACnet Datatypes/ST_BACnet_EventTransitionBits
TYPE ST_BACnet_EventTransitionBits:
STRUCT
	to_offnormal : BOOL;
	to_fault : BOOL;
	to_normal : BOOL;
END_STRUCT
END_TYPE

// Data types/BACnet Datatypes/ST_BACnet_ExceptionScheduleBool
TYPE ST_BACnet_ExceptionScheduleBool :
STRUCT
	bReqGet		: BOOL; (* set TRUE if property should reloaded, TRUE --> FALSE = request accepted (starting reload) *)
	bReqSet		: BOOL; (* set TRUE for property write request, TRUE --> FALSE = request accepted (starting storage) *)
	nGet		: USINT; (* reload counter, count up if property was loaded successful *)
	nSet		: USINT; (* save counter, count up if property was stored successful *)
	bBusy		: BOOL; (* started writing data into "arrEntries", don't write data to avoid concurrent access *)
	arrEntries	: ARRAY[0..BACnet_MaxExSchEntries] OF ST_BACnet_ExceptionScheduleEntryBool;
END_STRUCT
END_TYPE

// Data types/BACnet Datatypes/ST_BACnet_ExceptionScheduleEntryBool
TYPE ST_BACnet_ExceptionScheduleEntryBool :
STRUCT
	eEntryType		: E_BACnetCalendarEntryType;
	ePriority		: E_BACnetPriority;
	stDate			: ST_BACnet_ExceptionScheduleCalDate; (* date / date range *)
	stWeekNDay		: ST_BACnet_ExceptionScheduleCalWnD; (* week and day *)
	stCalRef		: ST_BACnet_ExceptionScheduleCalRef; (* week and day *)
	arrTimeValue	: ARRAY[0..BACnet_MaxTimeValues] OF ST_BACnet_TimeValueBool;
END_STRUCT
END_TYPE

// Data types/BACnet Datatypes/ST_BACnet_ExceptionScheduleEntryReal
TYPE ST_BACnet_ExceptionScheduleEntryReal :
STRUCT
	eEntryType		: E_BACnetCalendarEntryType;
	ePriority		: E_BACnetPriority;
	stDate			: ST_BACnet_ExceptionScheduleCalDate; (* date / date range *)
	stWeekNDay		: ST_BACnet_ExceptionScheduleCalWnD; (* week and day *)
	stCalRef		: ST_BACnet_ExceptionScheduleCalRef; (* week and day *)
	arrTimeValue	: ARRAY[0..BACnet_MaxTimeValues] OF ST_BACnet_TimeValueReal;
END_STRUCT
END_TYPE

// Data types/BACnet Datatypes/ST_BACnet_ExceptionScheduleReal
TYPE ST_BACnet_ExceptionScheduleReal :
STRUCT
	bReqGet		: BOOL; (* set TRUE if property should reloaded, TRUE --> FALSE = request accepted (starting reload) *)
	bReqSet		: BOOL; (* set TRUE for property write request, TRUE --> FALSE = request accepted (starting storage) *)
	nGet		: USINT; (* reload counter, count up if property was loaded successful *)
	nSet		: USINT; (* save counter, count up if property was stored successful *)
	bBusy		: BOOL; (* started writing data into "arrEntries", don't write data to avoid concurrent access *)
	arrEntries	: ARRAY[0..BACnet_MaxExSchEntries] OF ST_BACnet_ExceptionScheduleEntryReal;
END_STRUCT
END_TYPE

// Data types/BACnet Datatypes/ST_BACnet_LimitEnable
TYPE ST_BACnet_LimitEnable:
STRUCT
	lowLimitEnable : BOOL;
	highLimitEnable : BOOL;
END_STRUCT
END_TYPE

// Data types/BACnet Datatypes/ST_BACnet_LogBufferEntryReal
TYPE ST_BACnet_LogBufferEntryReal :
STRUCT
	nTimeStamp	: DWORD; (* 100ms since 1900 *)
	stDateTime	: ST_BACnet_DateTime; (* BACnet time stamp *)
	fValue		: REAL;
END_STRUCT
END_TYPE

// Data types/BACnet Datatypes/ST_BACnet_LogBufferReal
TYPE ST_BACnet_LogBufferReal :
STRUCT
	nGet		: USINT; (* Update date counter *)
	sObjectDesc	: T_MAXSTRING; (* Object description *)
	nCount		: UDINT; (* log buffer entries *)
	arrEntries	: ARRAY[0..BACnet_MaxLogBufferEntries] OF ST_BACnet_LogBufferEntryReal;
END_STRUCT
END_TYPE

// Data types/BACnet Datatypes/ST_BACnet_NSinkEvent
TYPE ST_BACnet_NSinkEvent :
STRUCT
	stValidFields	: ST_BACnet_NSinkEventValidFields;
	nProcessID		: UDINT;
	nDeviceID		: UDINT;
	tObjectID		: T_BACnet_ObjectIdentifier;
	stDateTime		: ST_BACnet_DateTime;
	nNC				: UDINT;	(* Notification class object instance *)
	nPriotity		: UDINT;
	eEventType		: E_BACNETEVENTTYPE;
	eNotifyType 	: E_BACNETNOTIFYTYPE;
	eFromState		: E_BACNETEVENTSTATE;
	eToState		: E_BACNETEVENTSTATE;
	sMessage		: T_MaxString;
	bAcknReq		: BOOL; (* Acknowledge required *)
END_STRUCT
END_TYPE

// Data types/BACnet Datatypes/ST_BACnet_ObjectIdentifierList
TYPE ST_BACnet_ObjectIdentifierList :
STRUCT
	nEntries	: UDINT;
	arrObjList	: ARRAY[0..BACnet_MaxObjIdList] OF T_BACnet_ObjectIdentifier :=[ 16#FFFFFFFF];
END_STRUCT
END_TYPE

// Data types/BACnet Datatypes/ST_BACnet_ObjectTypesSupported
TYPE ST_BACnet_ObjectTypesSupported:
STRUCT
	SuppAnalogInput : BOOL;
	SuppAnalogOutput : BOOL;
	SuppAnalogValue : BOOL;
	SuppBinaryInput : BOOL;
	SuppBinaryOutput : BOOL;
	SuppBinaryValue : BOOL;
	SuppCalendar : BOOL;
	SuppCommand : BOOL;
	SuppDevice : BOOL;
	SuppEventEnrollment : BOOL;
	SuppFile : BOOL;
	SuppGroup : BOOL;
	SuppLoop : BOOL;
	SuppMultiStateInput : BOOL;
	SuppMultiStateOutput : BOOL;
	SuppNotificationClass : BOOL;
	SuppProgram : BOOL;
	SuppSchedule : BOOL;
	SuppAveraging : BOOL;
	SuppMultiStateValue : BOOL;
	SuppTrendLog : BOOL;
	SuppLifeSafetyPoint : BOOL;
	SuppLifeSafetyZone : BOOL;
END_STRUCT
END_TYPE

// Data types/BACnet Datatypes/ST_BACnet_ProgramHandshakeRequests
TYPE ST_BACnet_ProgramHandshakeRequests :
STRUCT
	bLoad	: BOOL;
	bSetup	: BOOL;
	bRun	: BOOL;
	bHalt	: BOOL;
	bUnload	: BOOL;
END_STRUCT
END_TYPE

// Data types/BACnet Datatypes/ST_BACnet_ProgramHandshakeStates
TYPE ST_BACnet_ProgramHandshakeStates :
STRUCT
	bIdle		: BOOL;
	bLoading	: BOOL;
	bRunning	: BOOL;
	bWaiting	: BOOL;
	bHalted		: BOOL;
	bUnloading	: BOOL;
END_STRUCT
END_TYPE

// Data types/BACnet Datatypes/ST_BACnet_RecipientListDevice
TYPE ST_BACnet_RecipientListDevice :
STRUCT
	nEntries	: INT;
	arrDestList	: ARRAY[0..BACnet_MaxDestinationArray] OF ST_BACnet_RecipientListDeviceEntry;
END_STRUCT
END_TYPE

// Data types/BACnet Datatypes/ST_BACnet_RecipientListDeviceEntry
TYPE ST_BACnet_RecipientListDeviceEntry :
STRUCT
	bMonday		: BOOL := TRUE;
	bTuesday	: BOOL := TRUE;
	bWednesday	: BOOL := TRUE;
	bThursday	: BOOL := TRUE;
	bFriday		: BOOL := TRUE;
	bSaturday	: BOOL := TRUE;
	bSunday		: BOOL := TRUE;
	stFromTime	: ST_BACnet_Time :=
		(nHour		:= 0,
		nMinute		:= 0,
		nSecond		:= 0,
		nHundredths := 0);
	stToTime	: ST_BACnet_Time :=
		(nHour		:= 23,
		nMinute		:= 59,
		nSecond		:= 59,
		nHundredths := 99);
	tDeviceId	: T_BACnet_ObjectIdentifier := 16#FFFFFFFF;
	nProcessId	: UDINT;
	bToOffNormal: BOOL := TRUE;
	bToFault	: BOOL := TRUE;
	bToNormal	: BOOL := TRUE;
	bIssueConfirmedNotification	: BOOL;
END_STRUCT
END_TYPE

// Data types/BACnet Datatypes/ST_BACnet_ServicesSupported
TYPE ST_BACnet_ServicesSupported:
STRUCT
	SuppAcknowledgeAlarm : BOOL;
	SuppConfirmedCOVNotification : BOOL;
	SuppConfirmedEventNotification : BOOL;
	SuppGetAlarmSummary : BOOL;
	SuppGetEnrollmentSummary : BOOL;
	SuppSubscribeCOV : BOOL;
	SuppAtomicReadFile : BOOL;
	SuppAtomicWriteFile : BOOL;
	SuppAddListElement : BOOL;
	SuppRemoveListElement : BOOL;
	SuppCreateObject : BOOL;
	SuppDeleteObject : BOOL;
	SuppReadProperty : BOOL;
	SuppReadPropertyConditional : BOOL;
	SuppReadPropertyMultiple : BOOL;
	SuppWriteProperty : BOOL;
	SuppWritePropertyMultiple : BOOL;
	SuppDeviceCommunicationControl : BOOL;
	SuppConfirmedPrivateTransfer : BOOL;
	SuppConfirmedTextMessage : BOOL;
	SuppReinitializeDevice : BOOL;
	SuppVtOpen : BOOL;
	SuppVtClose : BOOL;
	SuppVtData : BOOL;
	SuppAuthenticate : BOOL;
	SuppRequestKey : BOOL;
	SuppIAm : BOOL;
	SuppIHave : BOOL;
	SuppUnconfirmedCOVNotification : BOOL;
	SuppUnconfirmedEventNotification : BOOL;
	SuppUnconfirmedPrivateTransfer : BOOL;
	SuppUnconfirmedTextMessage : BOOL;
	SuppTimeSynchronization : BOOL;
	SuppWhoHas : BOOL;
	SuppWhoIs : BOOL;
	SuppReadRange : BOOL;
	SuppUtcTimeSynchronization : BOOL;
	SuppLifeSafetyOperation : BOOL;
	SuppSubscribeCOVProperty : BOOL;
	SuppGetEventInformation : BOOL;
END_STRUCT
END_TYPE

// Data types/BACnet Datatypes/ST_BACnet_StatusFlags
TYPE ST_BACnet_StatusFlags:
STRUCT
	in_alarm : BOOL;
	fault : BOOL;
	overridden : BOOL;
	out_of_service : BOOL;
END_STRUCT
END_TYPE

// Data types/BACnet Datatypes/ST_BACnet_Time
TYPE ST_BACnet_Time :
STRUCT
	nHour		: BYTE := 16#FF; (* hour (0..23), (X'FF') = unspecified *)
	nMinute		: BYTE := 16#FF;	(* minute (0..59), (X'FF') = unspecified *)
	nSecond		: BYTE := 16#FF; (* (0..59), (X'FF') = unspecified *)
	nHundredths	: BYTE := 16#FF;	(* hundredths (0..99), (X'FF') = unspecified *)
END_STRUCT
END_TYPE

// Data types/BACnet Datatypes/ST_BACnet_TimeValue
TYPE ST_BACnet_TimeValue :
STRUCT
(*
	typedef struct _BACnetTimeValue
	{
	      BACnetTime time;
	      DWORD  reserved;  // 64bit Alignment
	      BACnetValue value;
	}BACnetTimeValue, *PBACnetTimeValue;
*)
	stTime	: ST_BACnet_Time;
	nRes	: DWORD;
	stValue	: ST_BACnet_Value;
END_STRUCT
END_TYPE

// Data types/BACnet Datatypes/ST_BACnet_TimeValueBool
TYPE ST_BACnet_TimeValueBool :
STRUCT
	bValid		: BOOL;
	stTime		: ST_BACnet_Time;
	eType		: E_BACnetDataTypes;
	bValue		: BOOL;
END_STRUCT
END_TYPE

// Data types/BACnet Datatypes/ST_BACnet_TimeValueList
TYPE ST_BACnet_TimeValueList :
STRUCT
(*
	typedef struct _BACnetTimeValueList
	{
	      DWORD nEntrySize; // 0x80000000 -> next entry
	      DWORD reserved;
	      BACnetTimeValue listEntry;
	}BACnetTimeValueList, *PBACnetTimeValueList;
*)
	nEntrySize	: DWORD;
	nRes		: DWORD;
	stListEntry	: ST_BACnet_TimeValue;
END_STRUCT
END_TYPE

// Data types/BACnet Datatypes/ST_BACnet_TimeValueReal
TYPE ST_BACnet_TimeValueReal :
STRUCT
	bValid		: BOOL;
	stTime		: ST_BACnet_Time;
	eType		: E_BACnetDataTypes;
	rValue		: REAL;
END_STRUCT
END_TYPE

// Data types/BACnet Datatypes/ST_BACnet_Value
TYPE ST_BACnet_Value :
STRUCT
(*
	typedef struct _BACnetValue  
	{
	      BACnetValueChoice choice;
	      DWORD                        length;     // Alignment + Datenlänge die folgt
	      union
	      {
	            BOOL                                     boolValue;
	            FLOAT                                    realValue;
	            DOUBLE                                   doubleValue;
	            INT                                      signedValue;
	            UINT                                     unsignedValue;
	            BYTE*                                    pOctedStringValue; 
	            CHAR*                                    pCharStringValue;
	            BACnetObjectIdentifier  objectIdentifierValue;
	            EnumerationValueType         enumerationValue;
	      };
	}BACnetValue, *PBACnetValue;
*)
	eValueChoice	: E_BACnetDataTypes;
	nRes1			: WORD; (* ENUM alignment *)
	cbData			: DWORD;
	nData			: BYTE;

END_STRUCT
END_TYPE

// Data types/BACnet Datatypes/ST_BACnet_WeeklyScheduleBool
TYPE ST_BACnet_WeeklyScheduleBool :
STRUCT
	bReqGet		: BOOL; (* set TRUE if property should reloaded, TRUE --> FALSE = request accepted (reload started) *)
	bReqSet		: BOOL; (* set TRUE for property write request, TRUE --> FALSE = request accepted (storage started) *)
	nGet		: USINT; (* reload counter, count up if property was loaded successful *)
	nSet		: USINT; (* save counter, count up if property was stored successful *)
	bBusy		: BOOL; (* started writing/reading data into/from "arrEntries", don't change data to avoid concurrent access *)
	arrEntries	: ARRAY[0..6] OF ARRAY[0..BACnet_MaxDayEntry] OF ST_BACnet_TimeValueBool;
END_STRUCT
END_TYPE

// Data types/BACnet Datatypes/ST_BACnet_WeeklyScheduleReal
TYPE ST_BACnet_WeeklyScheduleReal :
STRUCT
	bReqGet		: BOOL; (* set TRUE if property should reloaded, TRUE --> FALSE = request accepted (reload started) *)
	bReqSet		: BOOL; (* set TRUE for property write request, TRUE --> FALSE = request accepted (storage started) *)
	nGet		: USINT; (* reload counter, count up if property was loaded successful *)
	nSet		: USINT; (* save counter, count up if property was stored successful *)
	bBusy		: BOOL; (* started writing/reading data into/from "arrEntries", don't change data to avoid concurrent access *)
	arrEntries	: ARRAY[0..6] OF ARRAY[0..BACnet_MaxDayEntry] OF ST_BACnet_TimeValueReal;
END_STRUCT
END_TYPE

// Data types/BACnet Datatypes/T_BACnet_CalendarEntryTypeFilter
TYPE T_BACnet_CalendarEntryTypeFilter : ARRAY[0..4] OF E_BACnetCalendarEntryType; END_TYPE

// Data types/BACnet Datatypes/T_BACnet_ObjectIdentifier
TYPE T_BACnet_ObjectIdentifier : DWORD; END_TYPE

// Data types/BACnet Enumerations/E_BACNETACTION
TYPE E_BACNETACTION:
(
	BACnetAction_direct :=0,
	BACnetAction_reverse :=1
);
END_TYPE

// Data types/BACnet Enumerations/E_BACNETADAPTERSTATUS
TYPE E_BACNETADAPTERSTATUS :
(
	BACnetAdapterStatus_Init			:= 16#0,
	BACnetAdapterStatus_CheckIpAddr		:= 16#1,
	BACnetAdapterStatus_CheckParam		:= 16#2,
	BACnetAdapterStatus_GetGatewayMAC	:= 16#3,
	BACnetAdapterStatus_WaitGatewayMAC	:= 16#4,
	BACnetAdapterStatus_Complete		:= 16#8
);
END_TYPE

// Data types/BACnet Enumerations/E_BACNETBINARYPV
TYPE E_BACNETBINARYPV:
(
	BACnetBinaryPV_inactive :=0,
	BACnetBinaryPV_active :=1,
	BACnetBinaryPV_NULL := 2,
	BACnetBinaryPV_Nothing := 16#FFFF
);
END_TYPE

// Data types/BACnet Enumerations/E_BACNETDATATYPES
TYPE E_BACNETDATATYPES:
(
	BACnetDataType_Null :=0,
	BACnetDataType_Bool :=1,
	BACnetDataType_UnsignedInteger :=2,
	BACnetDataType_SignedInteger :=3,
	BACnetDataType_Real :=4,
	BACnetDataType_Double :=5,
	BACnetDataType_OctetString :=6,
	BACnetDataType_CharacterStringExt :=7,
	BACnetDataType_BitString :=8,
	BACnetDataType_Enumerated :=9,
	BACnetDataType_Date :=10,
	BACnetDataType_Time :=11,
	BACnetDataType_ObjectIdentifier :=12,
	BACnetDataType_DateTime :=14,
	BACnetDataType_ArrayIndex :=15,
	BACnetDataType_CalendarEntry :=16,
	BACnetDataType_ObjectType :=17,
	BACnetDataType_EventTransitionBits :=18,
	BACnetDataType_ActionList :=19,
	BACnetDataType_StatusFlags :=20,
	BACnetDataType_EventState :=21,
	BACnetDataType_Reliability :=22,
	BACnetDataType_Polarity :=23,
	BACnetDataType_EngineeringUnits :=25,
	BACnetDataType_PriorityValue :=26,
	BACnetDataType_LimitEnable :=27,
	BACnetDataType_NotifyType :=29,
	BACnetDataType_TimeStamp :=30,
	BACnetDataType_DeviceObjectPropertyReference :=31,
	BACnetDataType_DeviceStatus :=32,
	BACnetDataType_ServicesSupported :=33,
	BACnetDataType_ObjectTypesSupported :=34,
	BACnetDataType_Segmentation :=35,
	BACnetDataType_VTClass :=36,
	BACnetDataType_VTSession :=37,
	BACnetDataType_SessionKey :=38,
	BACnetDataType_Recipient :=39,
	BACnetDataType_AddressBinding :=40,
	BACnetDataType_COVSubscription :=41,
	BACnetDataType_EventType :=42,
	BACnetDataType_EventParameter :=43,
	BACnetDataType_FileAccessMethod :=44,
	BACnetDataType_ReadAccessSpecification :=45,
	BACnetDataType_ReadAccessResult :=46,
	BACnetDataType_ObjectPropertyReference :=47,
	BACnetDataType_SetpointReference :=48,
	BACnetDataType_Destination :=49,
	BACnetDataType_ProgramState :=50,
	BACnetDataType_ProgramRequest :=51,
	BACnetDataType_ProgramError :=52,
	BACnetDataType_DateRange :=53,
	BACnetDataType_DailySchedule :=54,
	BACnetDataType_SpecialEvent :=55,
	BACnetDataType_ClientCOV :=56,
	BACnetDataType_LogRecord :=57,
	BACnetDataType_LifeSafetyState :=58,
	BACnetDataType_LifeSafetyMode :=59,
	BACnetDataType_SilencedState :=60,
	BACnetDataType_LifeSafetyOperation :=61,
	BACnetDataType_BinaryPV :=62,
	BACnetDataType_DaysOfWeek :=63,
	BACnetDataType_WeekNDay :=64,
	BACnetDataType_TimeValue :=65,
	BACnetDataType_Value :=66,
	BACnetDataType_Address :=67,
	BACnetDataType_PropertyIdentifier :=68,
	BACnetDataType_EnumerationValueType :=69,
	BACnetDataType_BitFieldBit :=70,
	BACnetDataType_LogDatum :=71,
	BACnetDataType_AnyType :=72,
	BACnetDataType_PresentValue :=73,
	BACnetDataType_ContextTag :=74,
	BACnetDataType_ValueChoice :=75,
	BACnetDataType_LogStatus :=76,
	BACnetDataType_RecipientProcess :=77,
	BACnetDataType_SubscribeCOVPropertyRequest :=78,
	BACnetDataType_PropertyReference :=79,
	BACnetDataType_PropertyResult :=80,
	BACnetDataType_DeviceObjectPropertyValue :=81,
	BACnetDataType_COVNotificationRequest :=82,
	BACnetDataType_EventNotificationRequest :=83,
	BACnetDataType_NotificationParameters :=84,
	BACnetDataType_Change_of_Bitstring :=85,
	BACnetDataType_Change_of_State :=86,
	BACnetDataType_Change_of_Value :=87,
	BACnetDataType_Command_failure :=88,
	BACnetDataType_Floating_limit :=89,
	BACnetDataType_Out_of_Range :=90,
	BACnetDataType_PropertyValue :=91,
	BACnetDataType_Complex_Tag :=92,
	BACnetDataType_Change_of_life_safety :=93,
	BACnetDataType_Extended :=94,
	BACnetDataType_Buffer_ready :=95,
	BACnetDataType_Unsigned_range :=96,
	BACnetDataType_PropertyResultValue :=97,
	BACnetDataType_ServiceCOVPropSubscription :=98,
	BACnetDataType_ServiceCOVSubscription :=99,
	BACnetDataType_COVNotification :=100,
	BACnetDataType_AcknowledgeAlarmRequest :=101,
	BACnetDataType_VTOpenRequest :=102,
	BACnetDataType_Prescale :=103,
	BACnetDataType_Scale :=104,
	BACnetDataType_Action :=105,
	BACnetDataType_Error :=106,
	BACnetDataType_ErrorType :=107,
	BACnetDataType_ErrorClass :=108,
	BACnetDataType_ErrorCode :=109,
	BACnetDataType_RejectReason :=110,
	BACnetDataType_AbortReason :=111,
	BACnetDataType_BDTEntry :=112,
	BACnetDataType_IpEntry :=113,
	BACnetDataType_MaskEntry :=114,
	BACnetDataType_EthernetAddress := 115,
	BACnetDataType_LonTalkAddress := 116,
	BACnetDataType_LonTalkNeuronId := 117,
	BACnetDataType_NodeType := 118,
	BACnetDataType_DeviceObjectReference := 119,
	BACnetDataType_ActionCommand := 120,
	BACnetDataType_GetEventInformation := 121,
	BACnetDataType_GetEnrollmentSummaryCriteria := 122,
	BACnetDataType_GetEnrollmentSummaryCriteriaResponse := 123,
	BACnetDataType_DeviceCommunicationControl := 124,
	BACnetDataType_Int16 := 125,
	BACnetDataType_UInt16 := 126,
	BACnetDataType_UInt8 := 127,
	BACnetDataType_TypeInt8 := 128,
	BACnetDataType_Byte := 129,
	BACnetDataType_FDTEntry := 130,
	BACnetDataType_Address_3 := 131,
	BACnetDataType_Address_4 := 132,
	BACnetDataType_Address_5 := 133,
	BACnetDataType_PersistentDataState := 134,
	BACnetDataType_FallbackRealValue := 135,
	BACnetDataType_FallbackBinaryValue := 136,
	BACnetDataType_RealNull := 137, (* PresentValue in AnalogObj *)
	BACnetDataType_EnumeratedNull := 138, (* PresentValue in BinaryObj *)
	BACnetDataType_UnsignedIntegerNull := 139, (* PresentValue in Multistate *)
	BACnetDataType_Unknown := 140,
	BACnetDataType_DiagnosisPerformance := 200,
	BACnetDataType_DiagnosisEthStatistics := 201,
	BACnetDataType_FrameStatistics := 202,
	BACnetDataType_Info := 203,
	BACnetDataType_Diagnosis := 204,
	BACnetDataType_TcIoEthStatistic := 205,
	BACnetDataType_TcIoEthTxRxErrorCount := 206,
	BACnetDataType_TcIoEthPortStatistic := 207,
	BACnetDataType_ServerStatistics := 208,
	BACnetDataType_FrameServicesDiag := 209,
	BACnetDataType_UnsignedIntegerArr :=258,
	BACnetDataType_CharacterStringExtArr :=263,
	BACnetDataType_ObjectIdentifierArr :=268,
	BACnetDataType_CalendarEntryArr :=272,
	BACnetDataType_ActionListArr :=275,
	BACnetDataType_PriorityValueArr :=282,
	BACnetDataType_TimeStampArr :=286,
	BACnetDataType_DeviceObjectPropertyReferenceArr :=287,
	BACnetDataType_VTClassArr :=292,
	BACnetDataType_VTSessionArr :=293,
	BACnetDataType_SessionKeyArr :=294,
	BACnetDataType_RecipientArr :=295,
	BACnetDataType_AddressBindingArr :=296,
	BACnetDataType_COVSubscriptionArr :=297,
	BACnetDataType_ReadAccessSpecificationArr :=301,
	BACnetDataType_ReadAccessResultArr :=302,
	BACnetDataType_DestinationArr :=305,
	BACnetDataType_SpecialEventArr :=311,
	BACnetDataType_LogRecordArr :=313,
	BACnetDataType_LifeSafetyStateArr :=314,
	BACnetDataType_TimeValueArr :=321,
	BACnetDataType_UnsignedIntegerList :=514,
	BACnetDataType_CharacterStringExtList :=519,
	BACnetDataType_ReadAccessSpecificationList :=557,
	BACnetDataType_ReadAccessResultList :=558,
	BACnetDataType_SpecialEventList :=567,
	BACnetDataType_LogRecordList :=569,
	BACnetDataType_TimeValueList :=577,
	BACnetDataType_ValueList :=578,
	BACnetDataType_LogDatumList :=583,
	BACnetDataType_PropertyReferenceList :=591,
	BACnetDataType_PropertyResultList :=592,
	BACnetDataType_COVNotificationRequestList :=594,
	BACnetDataType_EventNotificationRequestList :=595,
	BACnetDataType_PropertyValueList :=603,
	BACnetDataType_DailyScheduleList :=1089
);
END_TYPE

// Data types/BACnet Enumerations/E_BACNETDAYSOFWEEKBITS
TYPE E_BACNETDAYSOFWEEKBITS :
(
	BACnetDaysOfWeekBits_Monday		:= 0,
	BACnetDaysOfWeekBits_Tuesday	:= 1,
	BACnetDaysOfWeekBits_Wednesday	:= 2,
	BACnetDaysOfWeekBits_Thursday	:= 3,
	BACnetDaysOfWeekBits_Friday		:= 4,
	BACnetDaysOfWeekBits_Saturday	:= 5,
	BACnetDaysOfWeekBits_Sunday		:= 6
);
END_TYPE

// Data types/BACnet Enumerations/E_BACNETDEVICESTATUS
TYPE E_BACNETDEVICESTATUS:
(
	BACnetDeviceStatus_Operational :=0,
	BACnetDeviceStatus_OperationalReadOnly :=1,
	BACnetDeviceStatus_DownloadRequired :=2,
	BACnetDeviceStatus_DownloadInProgress :=3,
	BACnetDeviceStatus_NonOperational :=4,
	BACnetDeviceStatus_BackupInProgress :=5
);
END_TYPE

// Data types/BACnet Enumerations/E_BACNETEVENTSTATE
TYPE E_BACNETEVENTSTATE:
(
	BACnetEventState_state_normal :=0,
	BACnetEventState_fault :=1,
	BACnetEventState_offnormal :=2,
	BACnetEventState_high_limit :=3,
	BACnetEventState_low_limit :=4,
	BACnetEventState_life_safety_alarm :=5
);
END_TYPE

// Data types/BACnet Enumerations/E_BACNETEVENTTRANSITIONBIT
TYPE E_BACNETEVENTTRANSITIONBIT:
(
	BACnetEventTransitionBit_to_offnormal :=0,
	BACnetEventTransitionBit_to_fault :=1,
	BACnetEventTransitionBit_to_normal :=2
);
END_TYPE

// Data types/BACnet Enumerations/E_BACNETEVENTTYPE
TYPE E_BACNETEVENTTYPE:
(
	BACnetEventType_change_of_bitstring :=0,
	BACnetEventType_change_of_state :=1,
	BACnetEventType_change_of_value :=2,
	BACnetEventType_command_failure :=3,
	BACnetEventType_floating_limit :=4,
	BACnetEventType_out_of_range :=5,
	BACnetEventType_complex_event_type :=6,
	BACnetEventType_deprecated7 :=7,
	BACnetEventType_change_of_life_safety :=8,
	BACnetEventType_enumeration :=9,
	BACnetEventType_buffer_ready :=10,
	BACnetEventType_unsigned_range :=11,
	BACnetEventType_reserved12 := 12,
	BACnetEventType_access_event := 13,
	BACnetEventType_double_out_of_range := 14,
	BACnetEventType_signed_out_of_range := 15,
	BACnetEventType_unsigned_out_of_range := 16,
	BACnetEventType_change_of_characterstring := 17,
	BACnetEventType_change_of_state_flags := 18
);
END_TYPE

// Data types/BACnet Enumerations/E_BACNETFILEACCESSMETHOD
TYPE E_BACNETFILEACCESSMETHOD:
(
	BACnetFileAccessMethod_record_access :=0,
	BACnetFileAccessMethod_stream_access :=1
);
END_TYPE

// Data types/BACnet Enumerations/E_BACNETLIFESAFETYMODE
TYPE E_BACNETLIFESAFETYMODE:
(
	BACnetLifeSafetyMode_off :=0,
	BACnetLifeSafetyMode_on :=1,
	BACnetLifeSafetyMode_test :=2,
	BACnetLifeSafetyMode_manned :=3,
	BACnetLifeSafetyMode_unmanned :=4,
	BACnetLifeSafetyMode_armed :=5,
	BACnetLifeSafetyMode_disarmed :=6,
	BACnetLifeSafetyMode_prearmed :=7,
	BACnetLifeSafetyMode_slow :=8,
	BACnetLifeSafetyMode_fast :=9,
	BACnetLifeSafetyMode_disconnected :=10,
	BACnetLifeSafetyMode_enabled :=11,
	BACnetLifeSafetyMode_disabled :=12,
	BACnetLifeSafetyMode_automatic_release_disabled :=13,
	BACnetLifeSafetyMode_mode_default :=14
);
END_TYPE

// Data types/BACnet Enumerations/E_BACNETLIFESAFETYOPERATION
TYPE E_BACNETLIFESAFETYOPERATION:
(
	BACnetLifeSafetyOperation_none :=0,
	BACnetLifeSafetyOperation_silence :=1,
	BACnetLifeSafetyOperation_silence_audible :=2,
	BACnetLifeSafetyOperation_silence_visual :=3,
	BACnetLifeSafetyOperation_reset :=4,
	BACnetLifeSafetyOperation_reset_alarm :=5,
	BACnetLifeSafetyOperation_reset_fault :=6,
	BACnetLifeSafetyOperation_unsilence := 7,
	BACnetLifeSafetyOperation_unsilence_audible := 8,
	BACnetLifeSafetyOperation_unsilence_visual := 9
);
END_TYPE

// Data types/BACnet Enumerations/E_BACNETLIMITENABLEBITS
TYPE E_BACNETLIMITENABLEBITS:
(
	BACnetLimitEnableBits_lowLimit :=0,
	BACnetLimitEnableBits_highLimit :=1
);
END_TYPE

// Data types/BACnet Enumerations/E_BACNETLOGGINGTYPE
TYPE E_BACNETLOGGINGTYPE :
(
	BACnetLoggingType_cov,
	BACnetLoggingType_polled,
	BACnetLoggingType_triggered
);
END_TYPE

// Data types/BACnet Enumerations/E_BACNETLOOPMODE
TYPE E_BACNETLOOPMODE :
(
	BACnetLoopMode_None,		(* LOOP object has unknown parameter settings *)
	BACnetLoopMode_Ideal,		(* Controller is in ideal form: P, I and D are in parallel junktion; unit of P, I and D is [1] (Kp, Ki, Kd) *)
	BACnetLoopMode_Standard		(* Controller works in standard form (most industrial applications): P parameter is applied to I and D; unit of I and D is time based [s] (Kp, Ti, Td) *)
);
END_TYPE

// Data types/BACnet Enumerations/E_BACNETNOTIFYTYPE
TYPE E_BACNETNOTIFYTYPE:
(
	BACnetNotifyType_alarm :=0,
	BACnetNotifyType_notify_event :=1,
	BACnetNotifyType_ack_notification :=2
);
END_TYPE

// Data types/BACnet Enumerations/E_BACNETOBJECTSUPPORTEDBITS
TYPE E_BACNETOBJECTSUPPORTEDBITS:
(
	BACnetObjectSupportedBits_AnalogInput :=0,
	BACnetObjectSupportedBits_AnalogOutput :=1,
	BACnetObjectSupportedBits_AnalogValue :=2,
	BACnetObjectSupportedBits_BinaryInput :=3,
	BACnetObjectSupportedBits_BinaryOutput :=4,
	BACnetObjectSupportedBits_BinaryValue :=5,
	BACnetObjectSupportedBits_Calendar :=6,
	BACnetObjectSupportedBits_Command :=7,
	BACnetObjectSupportedBits_Device :=8,
	BACnetObjectSupportedBits_EventEnrollment :=9,
	BACnetObjectSupportedBits_File :=10,
	BACnetObjectSupportedBits_Group :=11,
	BACnetObjectSupportedBits_Loop :=12,
	BACnetObjectSupportedBits_MultiStateInput :=13,
	BACnetObjectSupportedBits_MultiStateOutput :=14,
	BACnetObjectSupportedBits_NotificationClass :=15,
	BACnetObjectSupportedBits_Program :=16,
	BACnetObjectSupportedBits_Schedule :=17,
	BACnetObjectSupportedBits_Averaging :=18,
	BACnetObjectSupportedBits_MultiStateValue :=19,
	BACnetObjectSupportedBits_TrendLog :=20,
	BACnetObjectSupportedBits_LifeSafetyPoint :=21,
	BACnetObjectSupportedBits_LifeSafetyZone :=22,
	BACnetObjectSupportedBits_Accumulator := 23,
	BACnetObjectSupportedBits_PulseConverter := 24,
	BACnetObjectSupportedBits_EventLog := 25,
	BACnetObjectSupportedBits_GlobalGroup := 26,
	BACnetObjectSupportedBits_TrendLogMultiple := 27,
	BACnetObjectSupportedBits_LoadControl := 28,
	BACnetObjectSupportedBits_StructuredView := 29,
	BACnetObjectSupportedBits_AccessDoor := 30,
	BACnetObjectSupportedBits_unassigend31 := 31,
	BACnetObjectSupportedBits_AccessCredential := 32,
	BACnetObjectSupportedBits_AccessPoint := 33,
	BACnetObjectSupportedBits_AccessRights := 34,
	BACnetObjectSupportedBits_AccessUser := 35,
	BACnetObjectSupportedBits_AccessZone := 36,
	BACnetObjectSupportedBits_CredentialDataInput := 37,
	BACnetObjectSupportedBits_NetworkSecurity := 38,
	BACnetObjectSupportedBits_BitStringValue := 39,
	BACnetObjectSupportedBits_CharacterStringValue := 40,
	BACnetObjectSupportedBits_DatePatternValue := 41,
	BACnetObjectSupportedBits_DateValue := 42,
	BACnetObjectSupportedBits_DateTimePatternValue := 43,
	BACnetObjectSupportedBits_DateTimeValue := 44,
	BACnetObjectSupportedBits_IntegerValue := 45,
	BACnetObjectSupportedBits_LargeAnalogValue := 46,
	BACnetObjectSupportedBits_OctetStringValue := 47,
	BACnetObjectSupportedBits_PositiveIntegerValue := 48,
	BACnetObjectSupportedBits_TimePatternValue := 49,
	BACnetObjectSupportedBits_TimeValue := 50,
	BACnetObjectSupportedBits_NetworkPort := 51,
	BACnetObjectSupportedBits_AlertEnrollment := 52,
	BACnetObjectSupportedBits_Channel := 53
);
END_TYPE

// Data types/BACnet Enumerations/E_BACNETOBJECTTYPE
TYPE E_BACNETOBJECTTYPE:
(
	BACnetObjectType_AnalogInput :=0,
	BACnetObjectType_AnalogOutput :=1,
	BACnetObjectType_AnalogValue :=2,
	BACnetObjectType_BinaryInput :=3,
	BACnetObjectType_BinaryOutput :=4,
	BACnetObjectType_BinaryValue :=5,
	BACnetObjectType_Calendar :=6,
	BACnetObjectType_Command :=7,
	BACnetObjectType_Device :=8,
	BACnetObjectType_EventEnrollment :=9,
	BACnetObjectType_File :=10,
	BACnetObjectType_Group :=11,
	BACnetObjectType_Loop :=12,
	BACnetObjectType_MultiStateInput :=13,
	BACnetObjectType_MultiStateOutput :=14,
	BACnetObjectType_NotificationClass :=15,
	BACnetObjectType_Program :=16,
	BACnetObjectType_Schedule :=17,
	BACnetObjectType_Averaging :=18,
	BACnetObjectType_MultiStateValue :=19,
	BACnetObjectType_TrendLog :=20,
	BACnetObjectType_LifeSafetyPoint :=21,
	BACnetObjectType_LifeSafetyZone :=22,
	BACnetObjectType_Accumulator :=23,
	BACnetObjectType_PulseConverter :=24,
	BACnetObjectType_EventLog := 25,
	BACnetObjectType_GlobalGroup := 26,
	BACnetObjectType_TrendLogMultiple := 27,
	BACnetObjectType_LoadControl := 28,
	BACnetObjectType_StructuredView := 29,
	BACnetObjectType_AccessDoor := 30,
	BACnetObjectType_unassigend31 := 31,
	BACnetObjectType_AccessCredential := 32,
	BACnetObjectType_AccessPoint := 33,
	BACnetObjectType_AccessRights := 34,
	BACnetObjectType_AccessUser := 35,
	BACnetObjectType_AccessZone := 36,
	BACnetObjectType_CredentialDataInput := 37,
	BACnetObjectType_NetworkSecurity := 38,
	BACnetObjectType_BitStringValue := 39,
	BACnetObjectType_CharacterStringValue := 40,
	BACnetObjectType_DatePatternValue := 41,
	BACnetObjectType_DateValue := 42,
	BACnetObjectType_DateTimePatternValue := 43,
	BACnetObjectType_DateTimeValue := 44,
	BACnetObjectType_IntegerValue := 45,
	BACnetObjectType_LargeAnalogValue := 46,
	BACnetObjectType_OctetStringValue := 47,
	BACnetObjectType_PositiveIntegerValue := 48,
	BACnetObjectType_TimePatternValue := 49,
	BACnetObjectType_TimeValue := 50,
	BACnetObjectType_NetworkPort := 51,
	BACnetObjectType_AlertEnrollment := 52,
	BACnetObjectType_Channel := 53,


	(* keep at the end of list! *)
	BACnetObjectType_ZCount
);
END_TYPE

// Data types/BACnet Enumerations/E_BACNETPERSISTENTDATASTATE
TYPE E_BACNETPERSISTENTDATASTATE :
(
	BACnetPersistentData_Disabled,
	BACnetPersistentData_Initialize,
	BACnetPersistentData_NoChange,
	BACnetPersistentData_Ready,
	BACnetPersistentData_Write,
	BACnetPersistentData_Writing
);
END_TYPE

// Data types/BACnet Enumerations/E_BACNETPIDTUNINGMODE
TYPE E_BACNETPIDTUNINGMODE :
(
	BACnetPIDTuningMode_P,
	BACnetPIDTuningMode_PI,
	BACnetPIDTuningMode_PD,
	BACnetPIDTuningMode_PID
);
END_TYPE

// Data types/BACnet Enumerations/E_BACNETPOLARITY
TYPE E_BACNETPOLARITY:
(
	BACnetPolarity_normal :=0,
	BACnetPolarity_reverse :=1
);
END_TYPE

// Data types/BACnet Enumerations/E_BACNETPRIORITY
TYPE E_BACNETPRIORITY:
(
	BACnetPriority_None :=0,
	BACnetPriority_1 :=1,
	BACnetPriority_2 :=2,
	BACnetPriority_3 :=3,
	BACnetPriority_4 :=4,
	BACnetPriority_5 :=5,
	BACnetPriority_6 :=6,
	BACnetPriority_7 :=7,
	BACnetPriority_8 :=8,
	BACnetPriority_9 :=9,
	BACnetPriority_10 :=10,
	BACnetPriority_11 :=11,
	BACnetPriority_12 :=12,
	BACnetPriority_13 :=13,
	BACnetPriority_14 :=14,
	BACnetPriority_15 :=15,
	BACnetPriority_16 :=16
);
END_TYPE

// Data types/BACnet Enumerations/E_BACNETPROGRAMERROR
TYPE E_BACNETPROGRAMERROR:
(
	BACnetProgramError_program_normal :=0,
	BACnetProgramError_load_failed :=1,
	BACnetProgramError_progerror_internal :=2,
	BACnetProgramError_program :=3,
	BACnetProgramError_other :=4
);
END_TYPE

// Data types/BACnet Enumerations/E_BACNETPROGRAMREQUEST
TYPE E_BACNETPROGRAMREQUEST:
(
	BACnetProgramRequest_ready :=0,
	BACnetProgramRequest_load :=1,
	BACnetProgramRequest_run :=2,
	BACnetProgramRequest_halt :=3,
	BACnetProgramRequest_restart :=4,
	BACnetProgramRequest_unload :=5
);
END_TYPE

// Data types/BACnet Enumerations/E_BACNETPROGRAMSTATE
TYPE E_BACNETPROGRAMSTATE:
(
	BACnetProgramState_idle :=0,
	BACnetProgramState_loading :=1,
	BACnetProgramState_running :=2,
	BACnetProgramState_waiting :=3,
	BACnetProgramState_halted :=4,
	BACnetProgramState_unloading :=5
);
END_TYPE

// Data types/BACnet Enumerations/E_BACNETPROPERTYIDENTIFIER
TYPE E_BACNETPROPERTYIDENTIFIER:
(
	BACnetPropertyIdentifier_AckedTransitions 	:=	0	,
	BACnetPropertyIdentifier_AckRequired 	:=	1	,
	BACnetPropertyIdentifier_Action 	:=	2	,
	BACnetPropertyIdentifier_ActionText 	:=	3	,
	BACnetPropertyIdentifier_ActiveText 	:=	4	,
	BACnetPropertyIdentifier_ActiveVTSessions 	:=	5	,
	BACnetPropertyIdentifier_AlarmValue 	:=	6	,
	BACnetPropertyIdentifier_AlarmValues 	:=	7	,
	BACnetPropertyIdentifier_All 	:=	8	,
	BACnetPropertyIdentifier_AllWritesSuccessful 	:=	9	,
	BACnetPropertyIdentifier_ApduSegmentTimeout 	:=	10	,
	BACnetPropertyIdentifier_ApduTimeout 	:=	11	,
	BACnetPropertyIdentifier_ApplicationSoftwareVersion 	:=	12	,
	BACnetPropertyIdentifier_Archive 	:=	13	,
	BACnetPropertyIdentifier_Bias 	:=	14	,
	BACnetPropertyIdentifier_ChangeOfStateCount 	:=	15	,
	BACnetPropertyIdentifier_ChangeOfStateTime 	:=	16	,
	BACnetPropertyIdentifier_NotificationClass 	:=	17	,
	BACnetPropertyIdentifier_Reserved18 	:=	18	,
	BACnetPropertyIdentifier_ControlledVariableReference 	:=	19	,
	BACnetPropertyIdentifier_ControlledVariableUnits 	:=	20	,
	BACnetPropertyIdentifier_ControlledVariableValue 	:=	21	,
	BACnetPropertyIdentifier_CovIncrement 	:=	22	,
	BACnetPropertyIdentifier_DateList 	:=	23	,
	BACnetPropertyIdentifier_DaylightSavingsStatus 	:=	24	,
	BACnetPropertyIdentifier_Deadband 	:=	25	,
	BACnetPropertyIdentifier_DerivativeConstant 	:=	26	,
	BACnetPropertyIdentifier_DerivativeConstantUnits 	:=	27	,
	BACnetPropertyIdentifier_Description 	:=	28	,
	BACnetPropertyIdentifier_DescriptionOfHalt 	:=	29	,
	BACnetPropertyIdentifier_DeviceAddressBinding 	:=	30	,
	BACnetPropertyIdentifier_DeviceType 	:=	31	,
	BACnetPropertyIdentifier_EffectivePeriod 	:=	32	,
	BACnetPropertyIdentifier_ElapsedActiveTime 	:=	33	,
	BACnetPropertyIdentifier_ErrorLimit 	:=	34	,
	BACnetPropertyIdentifier_EventEnable 	:=	35	,
	BACnetPropertyIdentifier_EventState 	:=	36	,
	BACnetPropertyIdentifier_EventType 	:=	37	,
	BACnetPropertyIdentifier_ExceptionSchedule 	:=	38	,
	BACnetPropertyIdentifier_FaultValues 	:=	39	,
	BACnetPropertyIdentifier_FeedbackValue 	:=	40	,
	BACnetPropertyIdentifier_FileAccessMethod 	:=	41	,
	BACnetPropertyIdentifier_FileSize 	:=	42	,
	BACnetPropertyIdentifier_FileType 	:=	43	,
	BACnetPropertyIdentifier_FirmwareRevision 	:=	44	,
	BACnetPropertyIdentifier_HighLimit 	:=	45	,
	BACnetPropertyIdentifier_InactiveText 	:=	46	,
	BACnetPropertyIdentifier_InProcess 	:=	47	,
	BACnetPropertyIdentifier_InstanceOf 	:=	48	,
	BACnetPropertyIdentifier_IntegralConstant 	:=	49	,
	BACnetPropertyIdentifier_IntegralConstantUnits 	:=	50	,
	BACnetPropertyIdentifier_IssueConfirmedNotifications 	:=	51	,
	BACnetPropertyIdentifier_LimitEnable 	:=	52	,
	BACnetPropertyIdentifier_ListOfGroupMembers 	:=	53	,
	BACnetPropertyIdentifier_ListOfObjectPropertyReferences 	:=	54	,
	BACnetPropertyIdentifier_ListOfSessionKeys 	:=	55	,
	BACnetPropertyIdentifier_LocalDate 	:=	56	,
	BACnetPropertyIdentifier_LocalTime 	:=	57	,
	BACnetPropertyIdentifier_Location 	:=	58	,
	BACnetPropertyIdentifier_LowLimit 	:=	59	,
	BACnetPropertyIdentifier_ManipulatedVariableReference 	:=	60	,
	BACnetPropertyIdentifier_MaximumOutput 	:=	61	,
	BACnetPropertyIdentifier_MaxApduLengthAccepted 	:=	62	,
	BACnetPropertyIdentifier_MaxInfoFrames 	:=	63	,
	BACnetPropertyIdentifier_MaxMaster 	:=	64	,
	BACnetPropertyIdentifier_MaxPresValue 	:=	65	,
	BACnetPropertyIdentifier_MinimumOffTime 	:=	66	,
	BACnetPropertyIdentifier_MinimumOnTime 	:=	67	,
	BACnetPropertyIdentifier_MinimumOutput 	:=	68	,
	BACnetPropertyIdentifier_MinPresValue 	:=	69	,
	BACnetPropertyIdentifier_ModelName 	:=	70	,
	BACnetPropertyIdentifier_ModificationDate 	:=	71	,
	BACnetPropertyIdentifier_NotifyType 	:=	72	,
	BACnetPropertyIdentifier_NumberOfAPDURetries 	:=	73	,
	BACnetPropertyIdentifier_NumberOfStates 	:=	74	,
	BACnetPropertyIdentifier_ObjectIdentifier 	:=	75	,
	BACnetPropertyIdentifier_ObjectList 	:=	76	,
	BACnetPropertyIdentifier_ObjectName 	:=	77	,
	BACnetPropertyIdentifier_ObjectPropertyReference 	:=	78	,
	BACnetPropertyIdentifier_ObjectType 	:=	79	,
	BACnetPropertyIdentifier_Optional 	:=	80	,
	BACnetPropertyIdentifier_OutOfService 	:=	81	,
	BACnetPropertyIdentifier_OutputUnits 	:=	82	,
	BACnetPropertyIdentifier_EventParameters 	:=	83	,
	BACnetPropertyIdentifier_Polarity 	:=	84	,
	BACnetPropertyIdentifier_PresentValue 	:=	85	,
	BACnetPropertyIdentifier_Priority 	:=	86	,
	BACnetPropertyIdentifier_PriorityArray 	:=	87	,
	BACnetPropertyIdentifier_PriorityForWriting 	:=	88	,
	BACnetPropertyIdentifier_ProcessIdentifier 	:=	89	,
	BACnetPropertyIdentifier_ProgramChange 	:=	90	,
	BACnetPropertyIdentifier_ProgramLocation 	:=	91	,
	BACnetPropertyIdentifier_ProgramState 	:=	92	,
	BACnetPropertyIdentifier_ProportionalConstant 	:=	93	,
	BACnetPropertyIdentifier_ProportionalConstantUnits 	:=	94	,
	BACnetPropertyIdentifier_ProtocolConformanceClass 	:=	95	,
	BACnetPropertyIdentifier_ProtocolObjectTypesSupported 	:=	96	,
	BACnetPropertyIdentifier_ProtocolServicesSupported 	:=	97	,
	BACnetPropertyIdentifier_ProtocolVersion 	:=	98	,
	BACnetPropertyIdentifier_ReadOnly 	:=	99	,
	BACnetPropertyIdentifier_ReasonForHalt 	:=	100	,
	BACnetPropertyIdentifier_Recipient 	:=	101	,
	BACnetPropertyIdentifier_RecipientList 	:=	102	,
	BACnetPropertyIdentifier_Reliability 	:=	103	,
	BACnetPropertyIdentifier_RelinquishDefault 	:=	104	,
	BACnetPropertyIdentifier_Required 	:=	105	,
	BACnetPropertyIdentifier_Resolution 	:=	106	,
	BACnetPropertyIdentifier_SegmentationSupported 	:=	107	,
	BACnetPropertyIdentifier_Setpoint 	:=	108	,
	BACnetPropertyIdentifier_SetpointReference 	:=	109	,
	BACnetPropertyIdentifier_StateText 	:=	110	,
	BACnetPropertyIdentifier_StatusFlags 	:=	111	,
	BACnetPropertyIdentifier_SystemStatus 	:=	112	,
	BACnetPropertyIdentifier_TimeDelay 	:=	113	,
	BACnetPropertyIdentifier_TimeOfActiveTimeReset 	:=	114	,
	BACnetPropertyIdentifier_TimeOfStateCountReset 	:=	115	,
	BACnetPropertyIdentifier_TimeSynchronizationRecipients 	:=	116	,
	BACnetPropertyIdentifier_Units 	:=	117	,
	BACnetPropertyIdentifier_UpdateInterval 	:=	118	,
	BACnetPropertyIdentifier_UtcOffset 	:=	119	,
	BACnetPropertyIdentifier_VendorIdentifier 	:=	120	,
	BACnetPropertyIdentifier_VendorName 	:=	121	,
	BACnetPropertyIdentifier_VtClassesSupported 	:=	122	,
	BACnetPropertyIdentifier_WeeklySchedule 	:=	123	,
	BACnetPropertyIdentifier_AttemptedSamples 	:=	124	,
	BACnetPropertyIdentifier_AverageValue 	:=	125	,
	BACnetPropertyIdentifier_BufferSize 	:=	126	,
	BACnetPropertyIdentifier_ClientCovIncrement 	:=	127	,
	BACnetPropertyIdentifier_CovResubscriptionInterval 	:=	128	,
	BACnetPropertyIdentifier_CurrentNotifyTime 	:=	129	,
	BACnetPropertyIdentifier_EventTimeStamps 	:=	130	,
	BACnetPropertyIdentifier_LogBuffer 	:=	131	,
	BACnetPropertyIdentifier_LogDeviceObjectProperty 	:=	132	,
	BACnetPropertyIdentifier_Enable 	:=	133	,
	BACnetPropertyIdentifier_LogInterval 	:=	134	,
	BACnetPropertyIdentifier_MaximumValue 	:=	135	,
	BACnetPropertyIdentifier_MinimumValue 	:=	136	,
	BACnetPropertyIdentifier_NotificationThreshold 	:=	137	,
	BACnetPropertyIdentifier_PreviousNotifyTime 	:=	138	,
	BACnetPropertyIdentifier_ProtocolRevision 	:=	139	,
	BACnetPropertyIdentifier_RecordsSinceNotification 	:=	140	,
	BACnetPropertyIdentifier_RecordCount 	:=	141	,
	BACnetPropertyIdentifier_StartTime 	:=	142	,
	BACnetPropertyIdentifier_StopTime 	:=	143	,
	BACnetPropertyIdentifier_StopWhenFull 	:=	144	,
	BACnetPropertyIdentifier_TotalRecordCount 	:=	145	,
	BACnetPropertyIdentifier_ValidSamples 	:=	146	,
	BACnetPropertyIdentifier_WindowInterval 	:=	147	,
	BACnetPropertyIdentifier_WindowSamples 	:=	148	,
	BACnetPropertyIdentifier_MaximumValueTimestamp 	:=	149	,
	BACnetPropertyIdentifier_MinimumValueTimestamp 	:=	150	,
	BACnetPropertyIdentifier_VarianceValue 	:=	151	,
	BACnetPropertyIdentifier_ActiveCovSubscriptions 	:=	152	,
	BACnetPropertyIdentifier_BackupFailureTimeout 	:=	153	,
	BACnetPropertyIdentifier_ConfigurationFiles 	:=	154	,
	BACnetPropertyIdentifier_DatabaseRevision 	:=	155	,
	BACnetPropertyIdentifier_DirectReading 	:=	156	,
	BACnetPropertyIdentifier_LastRestoreTime 	:=	157	,
	BACnetPropertyIdentifier_MaintenanceRequired 	:=	158	,
	BACnetPropertyIdentifier_MemberOf 	:=	159	,
	BACnetPropertyIdentifier_Mode 	:=	160	,
	BACnetPropertyIdentifier_OperationExpected 	:=	161	,
	BACnetPropertyIdentifier_Setting 	:=	162	,
	BACnetPropertyIdentifier_Silenced 	:=	163	,
	BACnetPropertyIdentifier_TrackingValue 	:=	164	,
	BACnetPropertyIdentifier_ZoneMembers 	:=	165	,
	BACnetPropertyIdentifier_LifeSafetyAlarmValues 	:=	166	,
	BACnetPropertyIdentifier_MaxSegmentsAccepted 	:=	167	,
	BACnetPropertyIdentifier_ProfileName 	:=	168	,
	BACnetPropertyIdentifier_AutoSlaveDiscovery 	:=	169	,
	BACnetPropertyIdentifier_ManualSlaveAddressBinding 	:=	170	,
	BACnetPropertyIdentifier_SlaveAddressBinding 	:=	171	,
	BACnetPropertyIdentifier_SlaveProxyEnable 	:=	172	,
	BACnetPropertyIdentifier_LastNotifyRecord 	:=	173	,
	BACnetPropertyIdentifier_ScheduleDefault 	:=	174	,
	BACnetPropertyIdentifier_AcceptedModes 	:=	175	,
	BACnetPropertyIdentifier_AdjustValue 	:=	176	,
	BACnetPropertyIdentifier_Count 	:=	177	,
	BACnetPropertyIdentifier_CountBeforeChange 	:=	178	,
	BACnetPropertyIdentifier_CountChangeTime 	:=	179	,
	BACnetPropertyIdentifier_CovPeriod 	:=	180	,
	BACnetPropertyIdentifier_InputReference 	:=	181	,
	BACnetPropertyIdentifier_LimitMonitoringInverval 	:=	182	,
	BACnetPropertyIdentifier_LoggingObject 	:=	183	,
	BACnetPropertyIdentifier_LoggingRecord 	:=	184	,
	BACnetPropertyIdentifier_Prescale 	:=	185	,
	BACnetPropertyIdentifier_PulseRate 	:=	186	,
	BACnetPropertyIdentifier_Scale 	:=	187	,
	BACnetPropertyIdentifier_ScaleFactor 	:=	188	,
	BACnetPropertyIdentifier_UpdateTime 	:=	189	,
	BACnetPropertyIdentifier_ValueBeforeChange 	:=	190	,
	BACnetPropertyIdentifier_ValueSet 	:=	191	,
	BACnetPropertyIdentifier_ValueChangeTime 	:=	192	,
	BACnetPropertyIdentifier_AlignIntervals 	:=	193	,
	BACnetPropertyIdentifier_GroupMemberNames 	:=	194	,
	BACnetPropertyIdentifier_IntervalOffset 	:=	195	,
	BACnetPropertyIdentifier_LastRestartReason 	:=	196	,
	BACnetPropertyIdentifier_LoggingType 	:=	197	,
	BACnetPropertyIdentifier_MemberStatusFlags 	:=	198	,
	BACnetPropertyIdentifier_NotificationPeriod 	:=	199	,
	BACnetPropertyIdentifier_PreviousNotifyRecord 	:=	200	,
	BACnetPropertyIdentifier_RequestedUpdateInterval 	:=	201	,
	BACnetPropertyIdentifier_RestartNotificationRecipients 	:=	202	,
	BACnetPropertyIdentifier_TimeOfDeviceRestart 	:=	203	,
	BACnetPropertyIdentifier_TimeSynchronizationInterval 	:=	204	,
	BACnetPropertyIdentifier_Trigger 	:=	205	,
	BACnetPropertyIdentifier_UTCTimeSynchronizationRecipients 	:=	206	,
	BACnetPropertyIdentifier_NodeSubtype 	:=	207	,
	BACnetPropertyIdentifier_NodeType 	:=	208	,
	BACnetPropertyIdentifier_StructuredObjectList 	:=	209	,
	BACnetPropertyIdentifier_SubordinateAnnotations 	:=	210	,
	BACnetPropertyIdentifier_SubordinateList 	:=	211	,
	BACnetPropertyIdentifier_ActualShedLevel 	:=	212	,
	BACnetPropertyIdentifier_DutyWindow 	:=	213	,
	BACnetPropertyIdentifier_ExpectedShedLevel 	:=	214	,
	BACnetPropertyIdentifier_FullDutyBaseline 	:=	215	,
	BACnetPropertyIdentifier_NodeSubtype216 	:=	216	,
	BACnetPropertyIdentifier_NodeType217 	:=	217	,
	BACnetPropertyIdentifier_RequestedShedLevel 	:=	218	,
	BACnetPropertyIdentifier_ShedDuration 	:=	219	,
	BACnetPropertyIdentifier_ShedLevelDescriptions 	:=	220	,
	BACnetPropertyIdentifier_ShedLevels 	:=	221	,
	BACnetPropertyIdentifier_StateDescription 	:=	222	,
	BACnetPropertyIdentifier_DoorAlarmState 	:=	226	,
	BACnetPropertyIdentifier_DoorExtendedPulseTime 	:=	227	,
	BACnetPropertyIdentifier_DoorMembers 	:=	228	,
	BACnetPropertyIdentifier_DoorOpenTooLongTime 	:=	229	,
	BACnetPropertyIdentifier_DoorPulseTime 	:=	230	,
	BACnetPropertyIdentifier_DoorStatus 	:=	231	,
	BACnetPropertyIdentifier_DoorUnlockDelayTime 	:=	232	,
	BACnetPropertyIdentifier_LockStatus 	:=	233	,
	BACnetPropertyIdentifier_MaskedAlarmValues 	:=	234	,
	BACnetPropertyIdentifier_SecuredStatus 	:=	235	,
	BACnetPropertyIdentifier_BackupAndRestoreState 	:=	338	,
	BACnetPropertyIdentifier_BackupPreparationTime 	:=	339	,
	BACnetPropertyIdentifier_RestoreCompletionTime 	:=	340	,
	BACnetPropertyIdentifier_RestorePreparationTime 	:=	341	,
	BACnetPropertyIdentifier_EventMessageTexts 	:=	351	,
	BACnetPropertyIdentifier_EventMessageTextsConfig 	:=	352	,
	BACnetPropertyIdentifier_ScaleOffset 	:=	512	,
	BACnetPropertyIdentifier_IoBusNr 	:=	513	,
	BACnetPropertyIdentifier_IoModuleNr 	:=	514	,
	BACnetPropertyIdentifier_IoModuleChn 	:=	515	,
	BACnetPropertyIdentifier_PersistentData 	:=	516	,
	BACnetPropertyIdentifier_CurrentlyActivePriority 	:=	517	,
	BACnetPropertyIdentifier_LastConfirmedServiceAccess 	:=	518	,
	BACnetPropertyIdentifier_DataRequestMode 	:=	519	,
	BACnetPropertyIdentifier_DataRequestCycle 	:=	520	,
	BACnetPropertyIdentifier_FileName 	:=	521
);
END_TYPE

// Data types/BACnet Enumerations/E_BACNETRELIABILITY
TYPE E_BACNETRELIABILITY:
(
	BACnetReliability_no_fault_detected :=0,
	BACnetReliability_no_sensor :=1,
	BACnetReliability_over_range :=2,
	BACnetReliability_under_range :=3,
	BACnetReliability_open_loop :=4,
	BACnetReliability_shorted_loop :=5,
	BACnetReliability_no_output :=6,
	BACnetReliability_unreliable_other :=7,
	BACnetReliability_process_error :=8,
	BACnetReliability_multi_state_fault :=9,
	BACnetReliability_configuration_error :=10,
	BACnetReliability_reserved11 :=11,
	BACnetReliability_communication_failure :=12,
	BACnetReliability_member_fault :=13
);
END_TYPE

// Data types/BACnet Enumerations/E_BACNETSEGMENTATION
TYPE E_BACNETSEGMENTATION:
(
	BACnetSegmentation_both :=0,
	BACnetSegmentation_transmit :=1,
	BACnetSegmentation_receive :=2,
	BACnetSegmentation_no :=3
);
END_TYPE

// Data types/BACnet Enumerations/E_BACNETSERVICESSUPPORTEDBITS
TYPE E_BACNETSERVICESSUPPORTEDBITS:
(
	BACnetServiceSupportedBits_AcknowledgeAlarm :=0,
	BACnetServiceSupportedBits_ConfirmedCOVNotification :=1,
	BACnetServiceSupportedBits_ConfirmedEventNotification :=2,
	BACnetServiceSupportedBits_GetAlarmSummary :=3,
	BACnetServiceSupportedBits_GetEnrollmentSummary :=4,
	BACnetServiceSupportedBits_SubscribeCOV :=5,
	BACnetServiceSupportedBits_AtomicReadFile :=6,
	BACnetServiceSupportedBits_AtomicWriteFile :=7,
	BACnetServiceSupportedBits_AddListElement :=8,
	BACnetServiceSupportedBits_RemoveListElement :=9,
	BACnetServiceSupportedBits_CreateObject :=10,
	BACnetServiceSupportedBits_DeleteObject :=11,
	BACnetServiceSupportedBits_ReadProperty :=12,
	BACnetServiceSupportedBits_ReadPropertyConditional :=13,
	BACnetServiceSupportedBits_ReadPropertyMultiple :=14,
	BACnetServiceSupportedBits_WriteProperty :=15,
	BACnetServiceSupportedBits_WritePropertyMultiple :=16,
	BACnetServiceSupportedBits_DeviceCommunicationControl :=17,
	BACnetServiceSupportedBits_ConfirmedPrivateTransfer :=18,
	BACnetServiceSupportedBits_ConfirmedTextMessage :=19,
	BACnetServiceSupportedBits_ReinitializeDevice :=20,
	BACnetServiceSupportedBits_VtOpen :=21,
	BACnetServiceSupportedBits_VtClose :=22,
	BACnetServiceSupportedBits_VtData :=23,
	BACnetServiceSupportedBits_Authenticate :=24,
	BACnetServiceSupportedBits_RequestKey :=25,
	BACnetServiceSupportedBits_IAm :=26,
	BACnetServiceSupportedBits_IHave :=27,
	BACnetServiceSupportedBits_UnconfirmedCOVNotification :=28,
	BACnetServiceSupportedBits_UnconfirmedEventNotification :=29,
	BACnetServiceSupportedBits_UnconfirmedPrivateTransfer :=30,
	BACnetServiceSupportedBits_UnconfirmedTextMessage :=31,
	BACnetServiceSupportedBits_TimeSynchronization :=32,
	BACnetServiceSupportedBits_WhoHas :=33,
	BACnetServiceSupportedBits_WhoIs :=34,
	BACnetServiceSupportedBits_ReadRange :=35,
	BACnetServiceSupportedBits_UtcTimeSynchronization :=36,
	BACnetServiceSupportedBits_LifeSafetyOperation :=37,
	BACnetServiceSupportedBits_SubscribeCOVProperty :=38,
	BACnetServiceSupportedBits_GetEventInformation :=39
);
END_TYPE

// Data types/BACnet Enumerations/E_BACNETSILENCEDSTATE
TYPE E_BACNETSILENCEDSTATE:
(
	BACnetSilencedState_unsilenced :=0,
	BACnetSilencedState_audible_silenced :=1,
	BACnetSilencedState_visible_silenced :=2,
	BACnetSilencedState_all_silenced :=3
);
END_TYPE

// Data types/BACnet Enumerations/E_BACNETSTATUSFLAGS
TYPE E_BACNETSTATUSFLAGS:
(
	BACnetStatusFlags_in_alarm :=0,
	BACnetStatusFlags_fault :=1,
	BACnetStatusFlags_overridden :=2,
	BACnetStatusFlags_out_of_service :=3
);
END_TYPE

// Data types/BACnet Enumerations/E_BACNETSTRINGENCODINGTYPES
TYPE E_BACNETSTRINGENCODINGTYPES :
(
	BACnetStringEncodingTypes_AnsiUtf8	:= 0,
	BACnetStringEncodingTypes_DBCS		:= 1,
	BACnetStringEncodingTypes_JIS		:= 2,
	BACnetStringEncodingTypes_UCS4		:= 3,
	BACnetStringEncodingTypes_UCS2		:= 4,
	BACnetStringEncodingTypes_ISO8859	:= 5
);
END_TYPE

(*
---------------------------------------------
ISO8859
---------------------------------------------
						Part 1	Latin-1_ Western European__					
						Part 2	Latin-2_ Central European__					
						Part 3	Latin-3_ South European__					
						Part 4	Latin-4_ North European__					
Part 5	Latin/Cyrillic
Part 6	Latin/Arabic
Part 7	Latin/Greek
Part 8	Latin/Hebrew
						Part 9	Latin-5 _Turkish__					
						Part 10	Latin-6 _Nordic__					
Part 11	Latin/Thai
Part 12	"non-existent part" Latin/Devanagari
						Part 13	Latin-7_ Baltic Rim__					
						Part 14	Latin-8_ Celtic__					
Part 15	Latin-9
						Part 16	Latin-10_ South-Eastern European__					
---------------------------------------------
*)

